  MoveL 8360 to (2.11, -17.65, -15.61) mm, rotated rx -180 ry 0 rz 0.01 deg; joints [33.024, -56.054, 126.414, -145.496, 74.243, 170.404]
  MoveL 8361 to (-4.42, -18.62, -15.85) mm, rotated rx 180 ry 0 rz 0.01 deg; joints [32.823, -55.856, 126.015, -145.669, 74.039, 170.344]
  MoveL 8362 to (-6.16, -24.99, -16.1) mm, rotated rx 180 ry 0 rz 0.01 deg; joints [32.532, -55.905, 126.173, -145.984, 74.074, 170.492]
  MoveL 8363 to (-1.01, -29.13, -16.34) mm, rotated rx 180 ry 0 rz 0.01 deg; joints [32.498, -56.122, 126.697, -146.066, 74.322, 170.68]
  MoveL 8364 to (4.84, -26.08, -16.58) mm, rotated rx 180 ry 0 rz 0.01 deg; joints [32.765, -56.228, 126.959, -145.819, 74.501, 170.695]
  MoveL 8365 to (4.39, -19.49, -16.83) mm, rotated rx -180 ry 0 rz 0.01 deg; joints [33.011, -56.076, 126.643, -145.542, 74.41, 170.529]
  MoveL 8366 to (-1.82, -17.26, -17.07) mm, rotated rx -180 ry 0 rz 0.01 deg; joints [32.941, -55.829, 126.127, -145.571, 74.176, 170.391]
  MoveL 8367 to (-6.36, -22.07, -17.32) mm, rotated rx -180 ry 0 rz 0.01 deg; joints [32.641, -55.764, 126.029, -145.871, 74.092, 170.459]
  MoveL 8368 to (-3.77, -28.14, -17.56) mm, rotated rx -180 ry 0 rz 0.01 deg; joints [32.469, -55.939, 126.464, -146.088, 74.276, 170.66]
  MoveL 8369 to (2.83, -28.21, -17.8) mm, rotated rx 180 ry 0 rz 0.01 deg; joints [32.632, -56.125, 126.912, -145.963, 74.522, 170.765]
  MoveL 8370 to (5.54, -22.19, -18.05) mm, rotated rx 180 ry 0 rz 0.01 deg; joints [32.936, -56.08, 126.832, -145.648, 74.55, 170.659]
  MoveL 8371 to (1.11, -17.29, -18.29) mm, rotated rx -180 ry 0 rz 0.01 deg; joints [33.014, -55.839, 126.321, -145.525, 74.342, 170.478]
  MoveL 8372 to (-5.16, -19.39, -18.54) mm, rotated rx -180 ry 0 rz 0.01 deg; joints [32.776, -55.671, 125.99, -145.743, 74.162, 170.451]
  MoveL 8373 to (-5.74, -25.97, -18.78) mm, rotated rx 180 ry 0 rz 0.01 deg; joints [32.506, -55.758, 126.234, -146.043, 74.241, 170.62]
  MoveL 8374 to (0.05, -29.14, -19.02) mm, rotated rx 180 ry 0 rz 0.01 deg; joints [32.526, -55.976, 126.76, -146.07, 74.5, 170.793]
  MoveL 8375 to (5.28, -25.1, -19.27) mm, rotated rx 180 ry 0 rz 0.01 deg; joints [32.816, -56.044, 126.937, -145.792, 74.643, 170.775]
  MoveL 8376 to (3.68, -18.7, -19.51) mm, rotated rx 180 ry 0 rz 0.01 deg; joints [33.025, -55.862, 126.55, -145.547, 74.514, 170.596]
  MoveL 8377 to (-2.84, -17.6, -19.76) mm, rotated rx 180 ry 0 rz 0.01 deg; joints [32.904, -55.628, 126.064, -145.63, 74.283, 170.483]
  MoveL 8378 to (-6.45, -23.13, -20) mm, rotated rx -180 ry 0 rz 0.01 deg; joints [32.6, -55.604, 126.058, -145.944, 74.241, 170.581]
  MoveC 8379 to (-4.81, -27.09, -20) mm, rotated rx 180 ry 0 rz 0.01 deg; joints [32.486, -55.726, 126.34, -146.085, 74.352, 170.706] to (-0.84, -28.73, -20) mm, rotated rx 180 ry 0 rz 0.01 deg; joints [32.521, -55.876, 126.678, -146.079, 74.514, 170.805]
  MoveC 8380 to (3.12, -27.09, -20) mm, rotated rx 180 ry 0 rz 0.01 deg; joints [32.684, -55.967, 126.875, -145.929, 74.632, 170.821] to (4.76, -23.13, -20) mm, rotated rx 180 ry 0 rz 0.01 deg; joints [32.881, -55.944, 126.814, -145.722, 74.637, 170.744]
  MoveL 8381 to (4.76, -20.36, -20) mm, rotated rx 180 ry 0 rz 0.01 deg; joints [32.989, -55.893, 126.694, -145.602, 74.6, 170.673]
  MoveC 8382 to (3.66, -18.8, -20) mm, rotated rx 180 ry 0 rz 0.01 deg; joints [33.021, -55.83, 126.551, -145.556, 74.54, 170.617] to (1.82, -19.33, -20) mm, rotated rx -180 ry 0 rz 0.01 deg; joints [32.954, -55.785, 126.451, -145.615, 74.482, 170.604]
  MoveL 8383 to (-0.78, -22.57, -20) mm, rotated rx -180 ry 0 rz 0.01 deg; joints [32.763, -55.766, 126.417, -145.808, 74.434, 170.649]
  MoveC 8384 to (-1.01, -24.64, -20) mm, rotated rx -180 ry 0 rz 0.01 deg; joints [32.676, -55.797, 126.491, -145.903, 74.454, 170.699] to (0.75, -25.75, -20) mm, rotated rx 180 ry 0 rz 0.01 deg; joints [32.677, -55.871, 126.658, -145.917, 74.531, 170.753]
  MoveL 8385 to (2.65, -25.75, -20) mm, rotated rx -180 ry 0 rz 0.01 deg; joints [32.725, -55.928, 126.785, -145.879, 74.598, 170.78]
  MoveC 8386 to (4.14, -25.13, -20) mm, rotated rx -180 ry 0 rz 0.01 deg; joints [32.787, -55.962, 126.859, -145.822, 74.642, 170.786] to (4.76, -23.64, -20) mm, rotated rx -180 ry 0 rz 0.01 deg; joints [32.861, -55.953, 126.836, -145.745, 74.644, 170.757]
  MoveL 8387 to (4.76, -23.13, -20) mm, rotated rx -180 ry 0 rz 0.01 deg; joints [32.881, -55.944, 126.814, -145.722, 74.637, 170.744]
  MoveL 8388 to (3.55, -23.39, -20) mm, rotated rx 180 ry 0 rz 0.01 deg; joints [32.84, -55.912, 126.744, -145.758, 74.598, 170.733]
  MoveL 8389 to (4.04, -24.46, -20) mm, rotated rx 180 ry 0 rz 0.01 deg; joints [32.81, -55.946, 126.823, -145.795, 74.629, 170.767]
  MoveL 8390 to (4.24, -24.7, -20) mm, rotated rx -180 ry 0 rz 0.01 deg; joints [32.806, -55.957, 126.847, -145.802, 74.64, 170.776]
  MoveL 8391 to (8.68, -28.03, -20) mm, rotated rx 180 ry 0 rz 0.01 deg; joints [32.788, -56.151, 127.288, -145.858, 74.841, 170.925]
  MoveL 8392 to (9.37, -28.67, -20) mm, rotated rx 180 ry 0 rz 0.01 deg; joints [32.78, -56.184, 127.362, -145.872, 74.873, 170.951]
  MoveL 8393 to (9.68, -28.6, -20) mm, rotated rx -180 ry 0 rz 0.01 deg; joints [32.79, -56.192, 127.38, -145.863, 74.883, 170.954]
  MoveL 8394 to (10.02, -27.8, -20) mm, rotated rx 180 ry 0 rz 0.01 deg; joints [32.831, -56.188, 127.368, -145.821, 74.885, 170.939]
  MoveL 8395 to (10.22, -26.94, -20) mm, rotated rx -180 ry 0 rz 0.01 deg; joints [32.869, -56.178, 127.344, -145.779, 74.88, 170.92]
  MoveL 8396 to (10.27, -25.87, -20) mm, rotated rx -180 ry 0 rz 0.01 deg; joints [32.913, -56.16, 127.302, -145.731, 74.868, 170.893]
  MoveL 8397 to (10.27, 7.5, -20) mm, rotated rx -180 ry 0 rz 0.01 deg; joints [34.203, -55.533, 125.827, -144.284, 74.418, 170.028]
  MoveL 8398 to (6.2, -2.89, -20) mm, rotated rx -180 ry 0 rz 0.01 deg; joints [33.701, -55.609, 126.021, -144.814, 74.416, 170.241]
  MoveL 8399 to (5.98, -3.35, -20) mm, rotated rx -180 ry 0 rz 0.01 deg; joints [33.678, -55.611, 126.027, -144.839, 74.414, 170.25]
  MoveL 8400 to (1.99, -10.24, -20) mm, rotated rx 180 ry 0 rz 0.01 deg; joints [33.311, -55.62, 126.065, -145.217, 74.367, 170.371]
  MoveL 8401 to (1.7, -10.66, -20) mm, rotated rx -180 ry 0 rz 0.01 deg; joints [33.287, -55.62, 126.064, -145.241, 74.362, 170.378]
  MoveL 8402 to (-6.19, -20.5, -20) mm, rotated rx 180 ry 0 rz 0.01 deg; joints [32.708, -55.563, 125.963, -145.824, 74.216, 170.518]
  MoveL 8403 to (-6.61, -20.95, -20) mm, rotated rx -180 ry 0 rz 0.01 deg; joints [32.68, -55.558, 125.953, -145.852, 74.206, 170.523]
  MoveL 8404 to (-7.35, -21.58, -20) mm, rotated rx -180 ry 0 rz 0.01 deg; joints [32.638, -55.548, 125.931, -145.894, 74.189, 170.529]
  MoveL 8405 to (-7.68, -21.83, -20) mm, rotated rx 180 ry 0 rz 0.01 deg; joints [32.619, -55.542, 125.919, -145.912, 74.18, 170.53]
  MoveL 8406 to (-17.93, -28.66, -20) mm, rotated rx 180 ry 0 rz 0.01 deg; joints [32.101, -55.353, 125.516, -146.407, 73.906, 170.558]
  MoveL 8407 to (-18.59, -29, -20) mm, rotated rx 180 ry 0 rz 0.01 deg; joints [32.072, -55.339, 125.486, -146.434, 73.887, 170.557]
  MoveL 8408 to (-19.94, -29.53, -20) mm, rotated rx 180 ry 0 rz 0.01 deg; joints [32.019, -55.307, 125.416, -146.482, 73.845, 170.551]
  MoveL 8409 to (-20.23, -29.62, -20) mm, rotated rx -180 ry 0 rz 0.01 deg; joints [32.008, -55.3, 125.401, -146.492, 73.836, 170.549]
  MoveL 8410 to (-25.91, -31.27, -20) mm, rotated rx 180 ry 0 rz 0.01 deg; joints [31.807, -55.153, 125.082, -146.67, 73.654, 170.51]
  MoveL 8411 to (5.41, -31.27, -20) mm, rotated rx 180 ry 0 rz 0.01 deg; joints [32.578, -56.112, 127.208, -146.066, 74.769, 170.96]
  MoveL 8412 to (6.62, -31.07, -20) mm, rotated rx 180 ry 0 rz 0.01 deg; joints [32.616, -56.145, 127.281, -146.033, 74.809, 170.972]
  MoveL 8413 to (7.44, -30.76, -20) mm, rotated rx -180 ry 0 rz 0.01 deg; joints [32.649, -56.164, 127.323, -146.003, 74.834, 170.976]
  MoveL 8414 to (7.66, -30.63, -20) mm, rotated rx 180 ry 0 rz 0.01 deg; joints [32.66, -56.168, 127.332, -145.992, 74.84, 170.976]
  MoveL 8415 to (7.91, -29.14, -20) mm, rotated rx 180 ry 0 rz 0.01 deg; joints [32.724, -56.148, 127.284, -145.922, 74.828, 170.942]
  MoveL 8416 to (5.43, -26.15, -20) mm, rotated rx 180 ry 0 rz 0.01 deg; joints [32.779, -56.019, 126.989, -145.841, 74.701, 170.83]
  MoveL 8417 to (5.26, -25.18, -20) mm, rotated rx 180 ry 0 rz 0.01 deg; joints [32.813, -55.996, 126.936, -145.802, 74.682, 170.803]
  MoveL 8418 to (3.73, -18.75, -20.24) mm, rotated rx 180 ry 0 rz 0.01 deg; joints [33.025, -55.816, 126.554, -145.554, 74.555, 170.626]
  MoveL 8419 to (-2.76, -17.57, -20.49) mm, rotated rx 180 ry 0 rz 0.01 deg; joints [32.908, -55.581, 126.065, -145.634, 74.323, 170.51]
  MoveL 8420 to (-6.45, -23.04, -20.73) mm, rotated rx -180 ry 0 rz 0.01 deg; joints [32.603, -55.554, 126.052, -145.947, 74.278, 170.606]
  MoveL 8421 to (-2.92, -28.62, -20.98) mm, rotated rx 180 ry 0 rz 0.01 deg; joints [32.474, -55.747, 126.53, -146.124, 74.49, 170.808]
  MoveL 8422 to (3.61, -27.62, -21.22) mm, rotated rx -180 ry 0 rz 0.01 deg; joints [32.676, -55.91, 126.925, -145.953, 74.72, 170.886]
  MoveL 8423 to (5.31, -21.25, -21.46) mm, rotated rx 180 ry 0 rz 0.01 deg; joints [32.969, -55.828, 126.763, -145.642, 74.707, 170.757]
  MoveL 8424 to (0.16, -17.12, -21.71) mm, rotated rx -180 ry 0 rz 0.01 deg; joints [32.999, -55.58, 126.237, -145.568, 74.483, 170.585]
  MoveL 8425 to (-5.69, -20.19, -21.95) mm, rotated rx 180 ry 0 rz 0.01 deg; joints [32.734, -55.444, 125.975, -145.819, 74.33, 170.587]
  MoveL 8426 to (-5.22, -26.78, -22.2) mm, rotated rx 180 ry 0 rz 0.01 deg; joints [32.489, -55.562, 126.29, -146.099, 74.447, 170.771]
  MoveL 8427 to (1, -28.99, -22.44) mm, rotated rx -180 ry 0 rz 0.01 deg; joints [32.558, -55.774, 126.804, -146.076, 74.71, 170.927]
  MoveL 8428 to (5.52, -24.19, -22.68) mm, rotated rx -180 ry 0 rz 0.01 deg; joints [32.86, -55.807, 126.9, -145.778, 74.818, 170.88]
  MoveL 8429 to (2.94, -18.12, -22.93) mm, rotated rx -180 ry 0 rz 0.01 deg; joints [33.032, -55.601, 126.462, -145.567, 74.657, 170.695]
  MoveL 8430 to (-3.66, -18.05, -23.17) mm, rotated rx -180 ry 0 rz 0.01 deg; joints [32.869, -55.385, 126.014, -145.697, 74.435, 170.606]
  MoveL 8431 to (-6.38, -24.06, -23.41) mm, rotated rx 180 ry 0 rz 0.01 deg; joints [32.567, -55.397, 126.09, -146.014, 74.433, 170.729]
  MoveL 8432 to (-1.95, -28.96, -23.66) mm, rotated rx -180 ry 0 rz 0.01 deg; joints [32.486, -55.603, 126.598, -146.144, 74.668, 170.927]
  MoveL 8433 to (4.31, -26.88, -23.9) mm, rotated rx -180 ry 0 rz 0.01 deg; joints [32.725, -55.737, 126.93, -145.93, 74.875, 170.974]
  MoveL 8434 to (4.91, -20.31, -24.15) mm, rotated rx 180 ry 0 rz 0.01 deg; joints [32.997, -55.62, 126.685, -145.634, 74.819, 170.825]
  MoveL 8435 to (-0.86, -17.11, -24.39) mm, rotated rx 180 ry 0 rz 0.01 deg; joints [32.976, -55.372, 126.157, -145.612, 74.584, 170.667]
  MoveL 8436 to (-6.11, -21.12, -24.63) mm, rotated rx 180 ry 0 rz 0.01 deg; joints [32.689, -55.271, 125.976, -145.892, 74.465, 170.702]
  MoveL 8437 to (-4.54, -27.54, -24.88) mm, rotated rx 180 ry 0 rz 0.01 deg; joints [32.479, -55.418, 126.358, -146.143, 74.621, 170.897]
  MoveL 8438 to (1.96, -28.67, -25.12) mm, rotated rx 180 ry 0 rz 0.01 deg; joints [32.597, -55.618, 126.844, -146.066, 74.88, 171.03]
  MoveL 8439 to (5.62, -23.17, -25.37) mm, rotated rx -180 ry 0 rz 0.01 deg; joints [32.904, -55.611, 126.851, -145.755, 74.947, 170.953]
  MoveL 8440 to (2.04, -17.62, -25.61) mm, rotated rx 180 ry 0 rz 0.01 deg; joints [33.03, -55.387, 126.369, -145.587, 74.757, 170.767]
  MoveL 8441 to (-4.47, -18.67, -25.85) mm, rotated rx 180 ry 0 rz 0.01 deg; joints [32.826, -55.195, 125.975, -145.764, 74.552, 170.706]
  MoveL 8442 to (-6.13, -25.05, -26.1) mm, rotated rx -180 ry 0 rz 0.01 deg; joints [32.537, -55.245, 126.138, -146.077, 74.593, 170.854]
  MoveL 8443 to (-0.95, -29.14, -26.34) mm, rotated rx 180 ry 0 rz 0.01 deg; joints [32.506, -55.457, 126.662, -146.155, 74.846, 171.042]
  MoveL 8444 to (4.87, -26.03, -26.59) mm, rotated rx 180 ry 0 rz 0.01 deg; joints [32.774, -55.559, 126.919, -145.905, 75.023, 171.058]
  MoveL 8445 to (4.36, -19.45, -26.83) mm, rotated rx 180 ry 0 rz 0.01 deg; joints [33.019, -55.408, 126.599, -145.631, 74.927, 170.892]
  MoveL 8446 to (-1.87, -17.28, -27.07) mm, rotated rx -180 ry 0 rz 0.01 deg; joints [32.946, -55.166, 126.084, -145.663, 74.688, 170.753]
  MoveL 8447 to (-6.36, -22.11, -27.32) mm, rotated rx -180 ry 0 rz 0.01 deg; joints [32.646, -55.104, 125.99, -145.964, 74.607, 170.819]
  MoveL 8448 to (-3.74, -28.17, -27.56) mm, rotated rx 180 ry 0 rz 0.01 deg; joints [32.476, -55.275, 126.427, -146.178, 74.797, 171.02]
  MoveL 8449 to (2.87, -28.19, -27.8) mm, rotated rx 180 ry 0 rz 0.01 deg; joints [32.64, -55.456, 126.872, -146.051, 75.045, 171.127]
  MoveL 8450 to (5.54, -22.15, -28.05) mm, rotated rx -180 ry 0 rz 0.01 deg; joints [32.944, -55.411, 126.789, -145.736, 75.069, 171.023]
  MoveL 8451 to (1.08, -17.29, -28.29) mm, rotated rx -180 ry 0 rz 0.01 deg; joints [33.021, -55.174, 126.277, -145.616, 74.856, 170.841]
  MoveL 8452 to (-5.17, -19.41, -28.54) mm, rotated rx -180 ry 0 rz 0.01 deg; joints [32.781, -55.01, 125.948, -145.834, 74.675, 170.811]
  MoveL 8453 to (-5.73, -25.99, -28.78) mm, rotated rx -180 ry 0 rz 0.01 deg; joints [32.512, -55.095, 126.193, -146.133, 74.759, 170.979]
  MoveL 8454 to (0.07, -29.14, -29.02) mm, rotated rx -180 ry 0 rz 0.01 deg; joints [32.534, -55.308, 126.719, -146.158, 75.022, 171.154]
  MoveL 8455 to (5.29, -25.09, -29.27) mm, rotated rx -180 ry 0 rz 0.01 deg; joints [32.823, -55.374, 126.894, -145.88, 75.164, 171.138]
  MoveL 8456 to (3.67, -18.69, -29.51) mm, rotated rx 180 ry 0 rz 0.01 deg; joints [33.032, -55.195, 126.507, -145.636, 75.03, 170.96]
  MoveL 8457 to (-2.84, -17.6, -29.76) mm, rotated rx -180 ry 0 rz 0.01 deg; joints [32.911, -54.966, 126.021, -145.72, 74.796, 170.843]
  MoveL 8458 to (-6.45, -23.13, -30) mm, rotated rx -180 ry 0 rz 0.01 deg; joints [32.606, -54.941, 126.016, -146.033, 74.756, 170.939]
  MoveC 8459 to (-0.84, -28.74, -30) mm, rotated rx 180 ry 0 rz 0.01 deg; joints [32.527, -55.209, 126.635, -146.167, 75.034, 171.165] to (4.76, -23.13, -30) mm, rotated rx -180 ry 0 rz 0.01 deg; joints [32.887, -55.275, 126.771, -145.811, 75.156, 171.107]
  MoveL 8460 to (4.76, -20.36, -30) mm, rotated rx -180 ry 0 rz 0.01 deg; joints [32.995, -55.225, 126.651, -145.69, 75.117, 171.036]
  MoveC 8461 to (3.66, -18.8, -30) mm, rotated rx -180 ry 0 rz 0.01 deg; joints [33.028, -55.164, 126.509, -145.645, 75.056, 170.98] to (1.82, -19.33, -30) mm, rotated rx -180 ry 0 rz 0.01 deg; joints [32.961, -55.119, 126.408, -145.705, 74.998, 170.966]
  MoveL 8462 to (-0.77, -22.57, -30) mm, rotated rx 180 ry 0 rz 0.01 deg; joints [32.77, -55.1, 126.374, -145.897, 74.951, 171.01]
  MoveC 8463 to (-1.01, -24.64, -30) mm, rotated rx 180 ry 0 rz 0.01 deg; joints [32.683, -55.131, 126.448, -145.992, 74.971, 171.059] to (0.76, -25.75, -30) mm, rotated rx 180 ry 0 rz 0.01 deg; joints [32.684, -55.203, 126.615, -146.005, 75.05, 171.113]
  MoveL 8464 to (2.65, -25.75, -30) mm, rotated rx -180 ry 0 rz 0.01 deg; joints [32.731, -55.259, 126.742, -145.967, 75.117, 171.141]
  MoveC 8465 to (4.14, -25.14, -30) mm, rotated rx -180 ry 0 rz 0.01 deg; joints [32.793, -55.292, 126.816, -145.911, 75.162, 171.148] to (4.76, -23.64, -30) mm, rotated rx -180 ry 0 rz 0.01 deg; joints [32.867, -55.284, 126.793, -145.833, 75.163, 171.119]
  MoveL 8466 to (4.76, -23.13, -30) mm, rotated rx 180 ry 0 rz 0.01 deg; joints [32.887, -55.275, 126.771, -145.811, 75.156, 171.107]
  MoveL 8467 to (3.55, -23.4, -30) mm, rotated rx 180 ry 0 rz 0.01 deg; joints [32.846, -55.244, 126.701, -145.847, 75.116, 171.095]
  MoveL 8468 to (4.04, -24.46, -30) mm, rotated rx 180 ry 0 rz 0.01 deg; joints [32.817, -55.277, 126.78, -145.883, 75.149, 171.13]
  MoveL 8469 to (4.24, -24.7, -30) mm, rotated rx -180 ry 0 rz 0.01 deg; joints [32.813, -55.287, 126.804, -145.89, 75.159, 171.139]
  MoveL 8470 to (8.68, -28.03, -30) mm, rotated rx -180 ry 0 rz 0.01 deg; joints [32.794, -55.478, 127.245, -145.945, 75.364, 171.289]
  MoveL 8471 to (9.37, -28.67, -30) mm, rotated rx 180 ry 0 rz 0.01 deg; joints [32.787, -55.509, 127.318, -145.959, 75.397, 171.315]
  MoveL 8472 to (9.68, -28.6, -30) mm, rotated rx 180 ry 0 rz 0.01 deg; joints [32.797, -55.517, 127.336, -145.95, 75.407, 171.318]
  MoveL 8473 to (10.02, -27.8, -30) mm, rotated rx 180 ry 0 rz 0.01 deg; joints [32.837, -55.513, 127.325, -145.908, 75.408, 171.303]
  MoveL 8474 to (10.22, -26.94, -30) mm, rotated rx 180 ry 0 rz 0.01 deg; joints [32.876, -55.504, 127.301, -145.866, 75.403, 171.284]
  MoveL 8475 to (10.27, -25.87, -30) mm, rotated rx -180 ry 0 rz 0.01 deg; joints [32.92, -55.486, 127.258, -145.819, 75.39, 171.258]
  MoveL 8476 to (10.27, 7.47, -30) mm, rotated rx -180 ry 0 rz 0.01 deg; joints [34.208, -54.873, 125.786, -144.378, 74.921, 170.4]
  MoveL 8477 to (6.2, -2.89, -30) mm, rotated rx -180 ry 0 rz 0.01 deg; joints [33.707, -54.947, 125.978, -144.906, 74.923, 170.609]
  MoveL 8478 to (5.98, -3.35, -30) mm, rotated rx -180 ry 0 rz 0.01 deg; joints [33.684, -54.949, 125.984, -144.93, 74.922, 170.617]
  MoveL 8479 to (1.99, -10.24, -30) mm, rotated rx -180 ry 0 rz 0.01 deg; joints [33.317, -54.958, 126.022, -145.308, 74.877, 170.735]
  MoveL 8480 to (1.7, -10.66, -30) mm, rotated rx 180 ry 0 rz 0.01 deg; joints [33.294, -54.957, 126.021, -145.331, 74.873, 170.742]
  MoveL 8481 to (-6.17, -20.5, -30) mm, rotated rx -180 ry 0 rz 0.01 deg; joints [32.715, -54.902, 125.92, -145.914, 74.729, 170.876]
  MoveL 8482 to (-6.62, -20.95, -30) mm, rotated rx 180 ry 0 rz 0.01 deg; joints [32.687, -54.897, 125.91, -145.942, 74.72, 170.881]
  MoveL 8483 to (-7.36, -21.59, -30) mm, rotated rx 180 ry 0 rz 0.01 deg; joints [32.644, -54.887, 125.888, -145.984, 74.702, 170.886]
  MoveL 8484 to (-7.67, -21.83, -30) mm, rotated rx 180 ry 0 rz 0.01 deg; joints [32.626, -54.881, 125.877, -146.001, 74.694, 170.888]
  MoveL 8485 to (-17.71, -28.55, -30) mm, rotated rx 180 ry 0 rz 0.01 deg; joints [32.118, -54.7, 125.484, -146.487, 74.426, 170.909]
  MoveL 8486 to (-18.19, -28.82, -30) mm, rotated rx 180 ry 0 rz 0.01 deg; joints [32.096, -54.691, 125.463, -146.508, 74.412, 170.909]
  MoveL 8487 to (-19.2, -29.28, -30) mm, rotated rx 180 ry 0 rz 0.01 deg; joints [32.054, -54.668, 125.414, -146.547, 74.382, 170.906]
  MoveL 8488 to (-19.64, -29.44, -30) mm, rotated rx 180 ry 0 rz 0.01 deg; joints [32.036, -54.658, 125.391, -146.563, 74.368, 170.903]
  MoveL 8489 to (-25.81, -31.27, -30) mm, rotated rx -180 ry 0 rz 0.01 deg; joints [31.816, -54.503, 125.046, -146.758, 74.17, 170.858]
  MoveL 8490 to (5.41, -31.27, -30) mm, rotated rx 180 ry 0 rz 0.01 deg; joints [32.585, -55.439, 127.165, -146.153, 75.293, 171.321]
  MoveL 8491 to (6.62, -31.07, -30) mm, rotated rx 180 ry 0 rz 0.01 deg; joints [32.623, -55.471, 127.238, -146.12, 75.333, 171.335]
  MoveL 8492 to (7.44, -30.76, -30) mm, rotated rx 180 ry 0 rz 0.01 deg; joints [32.656, -55.49, 127.28, -146.09, 75.358, 171.339]
  MoveL 8493 to (7.66, -30.63, -30) mm, rotated rx -180 ry 0 rz 0.01 deg; joints [32.667, -55.494, 127.288, -146.079, 75.364, 171.339]
  MoveL 8494 to (7.91, -29.14, -30) mm, rotated rx -180 ry 0 rz 0.01 deg; joints [32.731, -55.475, 127.241, -146.009, 75.352, 171.305]
  MoveL 8495 to (5.43, -26.15, -30) mm, rotated rx -180 ry 0 rz 0.01 deg; joints [32.786, -55.348, 126.946, -145.929, 75.222, 171.193]
  MoveL 8496 to (5.26, -25.18, -30) mm, rotated rx 180 ry 0 rz 0.01 deg; joints [32.82, -55.326, 126.893, -145.89, 75.202, 171.166]
  MoveL 8497 to (3.74, -18.75, -30.24) mm, rotated rx 180 ry 0 rz 0.01 deg; joints [33.032, -55.149, 126.511, -145.643, 75.071, 170.989]
  MoveL 8498 to (-2.76, -17.57, -30.49) mm, rotated rx 180 ry 0 rz 0.01 deg; joints [32.914, -54.919, 126.022, -145.724, 74.835, 170.87]
  MoveL 8499 to (-6.45, -23.05, -30.73) mm, rotated rx -180 ry 0 rz 0.01 deg; joints [32.61, -54.891, 126.009, -146.036, 74.792, 170.963]
  MoveL 8500 to (-2.92, -28.62, -30.98) mm, rotated rx -180 ry 0 rz 0.01 deg; joints [32.481, -55.08, 126.486, -146.211, 75.009, 171.165]
  MoveL 8501 to (3.61, -27.62, -31.22) mm, rotated rx -180 ry 0 rz 0.01 deg; joints [32.683, -55.239, 126.881, -146.04, 75.241, 171.247]
  MoveL 8502 to (5.31, -21.25, -31.46) mm, rotated rx 180 ry 0 rz 0.01 deg; joints [32.976, -55.159, 126.719, -145.73, 75.224, 171.12]
  MoveL 8503 to (0.16, -17.13, -31.71) mm, rotated rx 180 ry 0 rz 0.01 deg; joints [33.006, -54.916, 126.192, -145.657, 74.996, 170.946]
  MoveL 8504 to (-5.69, -20.19, -31.95) mm, rotated rx -180 ry 0 rz 0.01 deg; joints [32.741, -54.782, 125.931, -145.908, 74.842, 170.945]
  MoveL 8505 to (-5.22, -26.78, -32.2) mm, rotated rx 180 ry 0 rz 0.01 deg; joints [32.496, -54.897, 126.245, -146.187, 74.963, 171.128]
  MoveL 8506 to (1, -29, -32.44) mm, rotated rx 180 ry 0 rz 0.01 deg; joints [32.565, -55.104, 126.759, -146.163, 75.23, 171.286]
  MoveL 8507 to (5.52, -24.19, -32.68) mm, rotated rx 180 ry 0 rz 0.01 deg; joints [32.867, -55.136, 126.854, -145.865, 75.336, 171.241]
  MoveL 8508 to (2.94, -18.12, -32.93) mm, rotated rx -180 ry 0 rz 0.01 deg; joints [33.038, -54.935, 126.416, -145.655, 75.171, 171.057]
  MoveL 8509 to (-3.66, -18.05, -33.17) mm, rotated rx 180 ry 0 rz 0.01 deg; joints [32.875, -54.722, 125.968, -145.785, 74.947, 170.964]
  MoveL 8510 to (-6.38, -24.06, -33.41) mm, rotated rx 180 ry 0 rz 0.01 deg; joints [32.574, -54.733, 126.044, -146.102, 74.946, 171.085]
  MoveL 8511 to (-1.95, -28.96, -33.66) mm, rotated rx 180 ry 0 rz 0.01 deg; joints [32.493, -54.935, 126.552, -146.23, 75.187, 171.284]
  MoveL 8512 to (4.31, -26.88, -33.9) mm, rotated rx -180 ry 0 rz 0.01 deg; joints [32.732, -55.066, 126.883, -146.016, 75.394, 171.335]
  MoveL 8513 to (4.91, -20.31, -34.15) mm, rotated rx 180 ry 0 rz 0.01 deg; joints [33.004, -54.95, 126.638, -145.72, 75.335, 171.187]
  MoveL 8514 to (-0.86, -17.12, -34.39) mm, rotated rx -180 ry 0 rz 0.01 deg; joints [32.982, -54.707, 126.11, -145.7, 75.096, 171.026]
  MoveL 8515 to (-6.11, -21.13, -34.63) mm, rotated rx -180 ry 0 rz 0.01 deg; joints [32.696, -54.608, 125.929, -145.98, 74.977, 171.058]
  MoveL 8516 to (-4.54, -27.54, -34.88) mm, rotated rx -180 ry 0 rz 0.01 deg; joints [32.485, -54.752, 126.31, -146.229, 75.137, 171.252]
  MoveL 8517 to (1.97, -28.67, -35.12) mm, rotated rx 180 ry 0 rz 0.01 deg; joints [32.603, -54.947, 126.796, -146.152, 75.399, 171.388]
  MoveL 8518 to (5.62, -23.17, -35.37) mm, rotated rx 180 ry 0 rz 0.01 deg; joints [32.911, -54.94, 126.803, -145.841, 75.464, 171.313]
  MoveL 8519 to (2.04, -17.62, -35.61) mm, rotated rx 180 ry 0 rz 0.01 deg; joints [33.037, -54.72, 126.321, -145.674, 75.269, 171.127]
  MoveL 8520 to (-4.47, -18.67, -35.85) mm, rotated rx -180 ry 0 rz 0.01 deg; joints [32.833, -54.531, 125.927, -145.851, 75.063, 171.063]
  MoveL 8521 to (-6.13, -25.06, -36.1) mm, rotated rx 180 ry 0 rz 0.01 deg; joints [32.543, -54.579, 126.089, -146.163, 75.106, 171.208]
  MoveL 8522 to (-0.95, -29.14, -36.34) mm, rotated rx 180 ry 0 rz 0.01 deg; joints [32.513, -54.787, 126.614, -146.24, 75.364, 171.398]
  MoveL 8523 to (4.87, -26.03, -36.59) mm, rotated rx 180 ry 0 rz 0.01 deg; joints [32.781, -54.886, 126.87, -145.99, 75.541, 171.418]
  MoveL 8524 to (4.36, -19.45, -36.83) mm, rotated rx 180 ry 0 rz 0.01 deg; joints [33.025, -54.739, 126.549, -145.717, 75.44, 171.253]
  MoveL 8525 to (-1.87, -17.28, -37.07) mm, rotated rx 180 ry 0 rz 0.01 deg; joints [32.953, -54.501, 126.035, -145.75, 75.198, 171.111]
  MoveL 8526 to (-6.36, -22.11, -37.32) mm, rotated rx 180 ry 0 rz 0.01 deg; joints [32.653, -54.439, 125.941, -146.05, 75.118, 171.173]
  MoveL 8527 to (-3.73, -28.17, -37.56) mm, rotated rx 180 ry 0 rz 0.01 deg; joints [32.482, -54.607, 126.377, -146.263, 75.312, 171.375]
  MoveL 8528 to (2.87, -28.19, -37.8) mm, rotated rx -180 ry 0 rz 0.01 deg; joints [32.647, -54.784, 126.822, -146.135, 75.563, 171.484]
  MoveL 8529 to (5.54, -22.16, -38.05) mm, rotated rx -180 ry 0 rz 0.01 deg; joints [32.95, -54.739, 126.739, -145.821, 75.584, 171.383]
  MoveL 8530 to (1.08, -17.29, -38.29) mm, rotated rx -180 ry 0 rz 0.01 deg; joints [33.027, -54.506, 126.227, -145.702, 75.366, 171.2]
  MoveL 8531 to (-5.17, -19.42, -38.54) mm, rotated rx -180 ry 0 rz 0.01 deg; joints [32.788, -54.345, 125.898, -145.92, 75.185, 171.166]
  MoveL 8532 to (-5.73, -25.99, -38.78) mm, rotated rx -180 ry 0 rz 0.01 deg; joints [32.519, -54.429, 126.143, -146.218, 75.272, 171.332]
  MoveL 8533 to (0.07, -29.14, -39.02) mm, rotated rx -180 ry 0 rz 0.01 deg; joints [32.54, -54.637, 126.668, -146.242, 75.539, 171.509]
  MoveL 8534 to (5.29, -25.1, -39.27) mm, rotated rx 180 ry 0 rz 0.01 deg; joints [32.83, -54.701, 126.843, -145.963, 75.68, 171.496]
  MoveL 8535 to (3.67, -18.7, -39.51) mm, rotated rx -180 ry 0 rz 0.01 deg; joints [33.039, -54.525, 126.456, -145.721, 75.542, 171.319]
  MoveL 8536 to (-2.84, -17.61, -39.76) mm, rotated rx 180 ry 0 rz 0.01 deg; joints [32.917, -54.3, 125.97, -145.806, 75.305, 171.199]
  MoveL 8537 to (-6.45, -23.13, -40) mm, rotated rx 180 ry 0 rz 0.01 deg; joints [32.613, -54.276, 125.964, -146.118, 75.266, 171.292]
  MoveC 8538 to (-0.84, -28.74, -40) mm, rotated rx 180 ry 0 rz 0.01 deg; joints [32.534, -54.537, 126.583, -146.251, 75.55, 171.519] to (4.76, -23.13, -40) mm, rotated rx 180 ry 0 rz 0.01 deg; joints [32.894, -54.602, 126.719, -145.895, 75.671, 171.465]
  MoveL 8539 to (4.76, -20.36, -40) mm, rotated rx -180 ry 0 rz 0.01 deg; joints [33.002, -54.553, 126.599, -145.775, 75.63, 171.395]
  MoveC 8540 to (3.66, -18.8, -40) mm, rotated rx -180 ry 0 rz 0.01 deg; joints [33.035, -54.494, 126.457, -145.729, 75.568, 171.339] to (1.82, -19.33, -40) mm, rotated rx 180 ry 0 rz 0.01 deg; joints [32.968, -54.45, 126.356, -145.789, 75.509, 171.323]
  MoveL 8541 to (-0.77, -22.57, -40) mm, rotated rx -180 ry 0 rz 0.01 deg; joints [32.777, -54.432, 126.323, -145.981, 75.463, 171.365]
  MoveC 8542 to (-1.01, -24.64, -40) mm, rotated rx -180 ry 0 rz 0.01 deg; joints [32.69, -54.461, 126.396, -146.076, 75.485, 171.414] to (0.76, -25.76, -40) mm, rotated rx -180 ry 0 rz 0.01 deg; joints [32.691, -54.532, 126.563, -146.089, 75.565, 171.469]
  MoveL 8543 to (2.65, -25.76, -40) mm, rotated rx 180 ry 0 rz 0.01 deg; joints [32.738, -54.587, 126.69, -146.051, 75.633, 171.498]
  MoveC 8544 to (4.15, -25.14, -40) mm, rotated rx 180 ry 0 rz 0.01 deg; joints [32.8, -54.619, 126.764, -145.994, 75.678, 171.505] to (4.76, -23.64, -40) mm, rotated rx 180 ry 0 rz 0.01 deg; joints [32.874, -54.611, 126.741, -145.917, 75.678, 171.478]
  MoveL 8545 to (4.76, -23.13, -40) mm, rotated rx -180 ry 0 rz 0.01 deg; joints [32.894, -54.602, 126.719, -145.895, 75.671, 171.465]
  MoveL 8546 to (3.55, -23.4, -40) mm, rotated rx 180 ry 0 rz 0.01 deg; joints [32.853, -54.572, 126.649, -145.931, 75.631, 171.453]
  MoveL 8547 to (4.04, -24.46, -40) mm, rotated rx 180 ry 0 rz 0.01 deg; joints [32.824, -54.605, 126.728, -145.967, 75.664, 171.487]
  MoveL 8548 to (4.24, -24.7, -40) mm, rotated rx -180 ry 0 rz 0.01 deg; joints [32.819, -54.614, 126.752, -145.973, 75.675, 171.496]
  MoveL 8549 to (8.68, -28.03, -40) mm, rotated rx -180 ry 0 rz 0.01 deg; joints [32.801, -54.801, 127.192, -146.028, 75.883, 171.648]
  MoveL 8550 to (9.37, -28.67, -40) mm, rotated rx -180 ry 0 rz 0.01 deg; joints [32.793, -54.832, 127.266, -146.042, 75.917, 171.674]
  MoveL 8551 to (9.68, -28.6, -40) mm, rotated rx 180 ry 0 rz 0.01 deg; joints [32.804, -54.839, 127.284, -146.033, 75.927, 171.677]
  MoveL 8552 to (10.02, -27.8, -40) mm, rotated rx 180 ry 0 rz 0.01 deg; joints [32.844, -54.835, 127.273, -145.991, 75.928, 171.663]
  MoveL 8553 to (10.22, -26.94, -40) mm, rotated rx 180 ry 0 rz 0.01 deg; joints [32.883, -54.826, 127.249, -145.949, 75.922, 171.644]
  MoveL 8554 to (10.27, -25.87, -40) mm, rotated rx 180 ry 0 rz 0.01 deg; joints [32.926, -54.809, 127.206, -145.901, 75.908, 171.618]
  MoveL 8555 to (10.27, 7.44, -40) mm, rotated rx 180 ry 0 rz 0.01 deg; joints [34.214, -54.21, 125.736, -144.467, 75.42, 170.767]
  MoveL 8556 to (6.19, -2.89, -40) mm, rotated rx 180 ry 0 rz 0.01 deg; joints [33.714, -54.282, 125.927, -144.993, 75.427, 170.972]
  MoveL 8557 to (5.98, -3.35, -40) mm, rotated rx 180 ry 0 rz 0.01 deg; joints [33.691, -54.284, 125.932, -145.016, 75.425, 170.98]
  MoveL 8558 to (1.99, -10.24, -40) mm, rotated rx -180 ry 0 rz 0.01 deg; joints [33.324, -54.293, 125.97, -145.394, 75.383, 171.095]
  MoveL 8559 to (1.7, -10.66, -40) mm, rotated rx 180 ry 0 rz 0.01 deg; joints [33.3, -54.292, 125.969, -145.417, 75.379, 171.101]
  MoveL 8560 to (-6.17, -20.49, -40) mm, rotated rx 180 ry 0 rz 0.01 deg; joints [32.722, -54.238, 125.869, -145.999, 75.239, 171.23]
  MoveL 8561 to (-6.61, -20.95, -40) mm, rotated rx 180 ry 0 rz 0.01 deg; joints [32.693, -54.233, 125.859, -146.027, 75.229, 171.234]
  MoveL 8562 to (-7.36, -21.59, -40) mm, rotated rx -180 ry 0 rz 0.01 deg; joints [32.65, -54.222, 125.836, -146.07, 75.211, 171.239]
  MoveL 8563 to (-7.67, -21.82, -40) mm, rotated rx -180 ry 0 rz 0.01 deg; joints [32.633, -54.217, 125.825, -146.086, 75.204, 171.24]
  MoveL 8564 to (-17.48, -28.43, -40) mm, rotated rx 180 ry 0 rz 0.01 deg; joints [32.135, -54.044, 125.443, -146.563, 74.942, 171.257]
  MoveL 8565 to (-17.94, -28.7, -40) mm, rotated rx -180 ry 0 rz 0.01 deg; joints [32.113, -54.035, 125.423, -146.583, 74.929, 171.256]
  MoveL 8566 to (-19.17, -29.27, -40) mm, rotated rx 180 ry 0 rz 0.01 deg; joints [32.061, -54.009, 125.363, -146.631, 74.892, 171.252]
  MoveL 8567 to (-19.62, -29.44, -40) mm, rotated rx -180 ry 0 rz 0.01 deg; joints [32.044, -53.998, 125.34, -146.647, 74.878, 171.249]
  MoveL 8568 to (-25.71, -31.27, -40) mm, rotated rx 180 ry 0 rz 0.01 deg; joints [31.825, -53.849, 125.002, -146.842, 74.681, 171.202]
  MoveL 8569 to (5.41, -31.27, -40) mm, rotated rx -180 ry 0 rz 0.01 deg; joints [32.591, -54.763, 127.112, -146.235, 75.812, 171.678]
  MoveL 8570 to (6.62, -31.07, -40) mm, rotated rx 180 ry 0 rz 0.01 deg; joints [32.629, -54.794, 127.185, -146.202, 75.853, 171.692]
  MoveL 8571 to (7.44, -30.76, -40) mm, rotated rx 180 ry 0 rz 0.01 deg; joints [32.662, -54.813, 127.227, -146.172, 75.878, 171.697]
  MoveL 8572 to (7.66, -30.63, -40) mm, rotated rx -180 ry 0 rz 0.01 deg; joints [32.673, -54.817, 127.236, -146.162, 75.884, 171.697]
  MoveL 8573 to (7.67, -29.55, -40) mm, rotated rx -180 ry 0 rz 0.01 deg; joints [32.716, -54.798, 127.191, -146.115, 75.869, 171.67]
  MoveL 8574 to (3.92, -27.15, -40) mm, rotated rx -180 ry 0 rz 0.01 deg; joints [32.715, -54.648, 126.835, -146.086, 75.699, 171.552]
  MoveL 8575 to (-0.53, -24.82, -40) mm, rotated rx 180 ry 0 rz 0.01 deg; joints [32.695, -54.478, 126.436, -146.074, 75.505, 171.426]
  MoveL 8576 to (-1.53, -24.26, -40) mm, rotated rx -180 ry 0 rz 0.01 deg; joints [32.692, -54.439, 126.344, -146.07, 75.46, 171.396]
  MoveL 8577 to (-1.89, -24.46, -40) mm, rotated rx 180 ry 0 rz 0.01 deg; joints [32.675, -54.432, 126.329, -146.086, 75.45, 171.395]
  MoveL 8578 to (1.29, -30.05, -40.24) mm, rotated rx 180 ry 0 rz 0.01 deg; joints [32.536, -54.606, 126.782, -146.267, 75.658, 171.593]
  MoveL 8579 to (7.7, -29.59, -40.47) mm, rotated rx 180 ry 0 rz 0.01 deg; joints [32.715, -54.768, 127.192, -146.12, 75.895, 171.689]
  MoveL 8580 to (10.06, -23.61, -40.71) mm, rotated rx 180 ry 0 rz 0.01 deg; joints [33.01, -54.715, 127.09, -145.813, 75.904, 171.584]
  MoveL 8581 to (5.69, -18.9, -40.95) mm, rotated rx 180 ry 0 rz 0.01 deg; joints [33.083, -54.49, 126.591, -145.7, 75.69, 171.406]
  MoveL 8582 to (-0.45, -20.81, -41.18) mm, rotated rx 180 ry 0 rz 0.01 deg; joints [32.854, -54.33, 126.261, -145.909, 75.51, 171.368]
  MoveL 8583 to (-1.38, -27.17, -41.42) mm, rotated rx 180 ry 0 rz 0.01 deg; joints [32.583, -54.399, 126.472, -146.205, 75.581, 171.521]
  MoveL 8584 to (3.96, -30.76, -41.66) mm, rotated rx 180 ry 0 rz 0.01 deg; joints [32.576, -54.6, 126.984, -146.256, 75.838, 171.702]
  MoveL 8585 to (9.5, -27.49, -41.89) mm, rotated rx -180 ry 0 rz 0.01 deg; joints [32.844, -54.686, 127.213, -146.003, 76.002, 171.715]
  MoveL 8586 to (8.94, -21.08, -42.13) mm, rotated rx 180 ry 0 rz 0.01 deg; joints [33.081, -54.542, 126.897, -145.738, 75.9, 171.554]
  MoveL 8587 to (2.92, -18.82, -42.37) mm, rotated rx 180 ry 0 rz 0.01 deg; joints [33.017, -54.314, 126.394, -145.764, 75.662, 171.412]
  MoveL 8588 to (-1.72, -23.27, -42.61) mm, rotated rx -180 ry 0 rz 0.01 deg; joints [32.727, -54.242, 126.274, -146.052, 75.572, 171.46]
  MoveL 8589 to (0.29, -29.38, -42.84) mm, rotated rx 180 ry 0 rz 0.01 deg; joints [32.539, -54.39, 126.671, -146.279, 75.746, 171.652]
  MoveL 8590 to (6.67, -30.2, -43.08) mm, rotated rx -180 ry 0 rz 0.01 deg; joints [32.667, -54.571, 127.133, -146.188, 76.001, 171.78]
  MoveL 8591 to (10.17, -24.81, -43.32) mm, rotated rx 180 ry 0 rz 0.01 deg; joints [32.967, -54.562, 127.134, -145.884, 76.06, 171.709]
  MoveL 8592 to (6.81, -19.32, -43.55) mm, rotated rx -180 ry 0 rz 0.01 deg; joints [33.097, -54.354, 126.67, -145.717, 75.87, 171.527]
  MoveL 8593 to (0.41, -19.98, -43.79) mm, rotated rx 180 ry 0 rz 0.01 deg; joints [32.91, -54.166, 126.268, -145.877, 75.661, 171.452]
  MoveL 8594 to (-1.75, -26.03, -44.03) mm, rotated rx -180 ry 0 rz 0.01 deg; joints [32.62, -54.193, 126.382, -146.184, 75.684, 171.579]
  MoveL 8595 to (2.77, -30.6, -44.26) mm, rotated rx 180 ry 0 rz 0.01 deg; joints [32.554, -54.386, 126.882, -146.294, 75.927, 171.771]
  MoveL 8596 to (8.85, -28.5, -44.5) mm, rotated rx -180 ry 0 rz 0.01 deg; joints [32.79, -54.508, 127.197, -146.081, 76.128, 171.822]
  MoveC 8597 to (7.97, -20.62, -44.5) mm, rotated rx 180 ry 0 rz 0.01 deg; joints [33.076, -54.346, 126.798, -145.757, 75.979, 171.612] to (0.09, -21.49, -44.5) mm, rotated rx -180 ry 0 rz 0.01 deg; joints [32.843, -54.135, 126.308, -145.954, 75.708, 171.51]
  MoveL 8598 to (-0.77, -22.57, -44.5) mm, rotated rx 180 ry 0 rz 0.01 deg; joints [32.78, -54.129, 126.296, -146.018, 75.692, 171.524]
  MoveC 8599 to (-1.01, -24.64, -44.5) mm, rotated rx 180 ry 0 rz 0.01 deg; joints [32.693, -54.159, 126.37, -146.113, 75.714, 171.572] to (0.76, -25.75, -44.5) mm, rotated rx 180 ry 0 rz 0.01 deg; joints [32.694, -54.229, 126.537, -146.125, 75.795, 171.627]
  MoveL 8600 to (2.65, -25.75, -44.5) mm, rotated rx 180 ry 0 rz 0.01 deg; joints [32.741, -54.283, 126.664, -146.087, 75.863, 171.657]
  MoveC 8601 to (4.14, -25.14, -44.5) mm, rotated rx 180 ry 0 rz 0.01 deg; joints [32.803, -54.315, 126.737, -146.03, 75.908, 171.665] to (4.76, -23.64, -44.5) mm, rotated rx 180 ry 0 rz 0.01 deg; joints [32.877, -54.307, 126.714, -145.953, 75.908, 171.637]
  MoveL 8602 to (4.76, -20.36, -44.5) mm, rotated rx -180 ry 0 rz 0.01 deg; joints [33.005, -54.25, 126.572, -145.811, 75.86, 171.555]
  MoveC 8603 to (3.66, -18.8, -44.5) mm, rotated rx -180 ry 0 rz 0.01 deg; joints [33.038, -54.191, 126.43, -145.766, 75.797, 171.498] to (1.82, -19.33, -44.5) mm, rotated rx 180 ry 0 rz 0.01 deg; joints [32.971, -54.147, 126.33, -145.826, 75.738, 171.483]
  MoveL 8604 to (0.09, -21.49, -44.5) mm, rotated rx -180 ry 0 rz 0.01 deg; joints [32.843, -54.135, 126.308, -145.954, 75.708, 171.51]
  MoveC 8605 to (-0.12, -22.22, -44.5) mm, rotated rx -180 ry 0 rz 0.01 deg; joints [32.809, -54.142, 126.325, -145.99, 75.711, 171.525] to (0.24, -22.89, -44.5) mm, rotated rx -180 ry 0 rz 0.01 deg; joints [32.792, -54.164, 126.378, -146.012, 75.734, 171.548]
  MoveL 8606 to (7.77, -29, -44.5) mm, rotated rx -180 ry 0 rz 0.01 deg; joints [32.743, -54.486, 127.147, -146.125, 76.096, 171.818]
  MoveL 8607 to (7.66, -30.63, -44.5) mm, rotated rx 180 ry 0 rz 0.01 deg; joints [32.676, -54.511, 127.21, -146.197, 76.117, 171.856]
  MoveL 8608 to (7.44, -30.76, -44.5) mm, rotated rx 180 ry 0 rz 0.01 deg; joints [32.665, -54.507, 127.201, -146.208, 76.111, 171.856]
  MoveL 8609 to (6.62, -31.07, -44.5) mm, rotated rx -180 ry 0 rz 0.01 deg; joints [32.633, -54.488, 127.159, -146.238, 76.086, 171.851]
  MoveL 8610 to (5.41, -31.27, -44.5) mm, rotated rx 180 ry 0 rz 0.01 deg; joints [32.594, -54.457, 127.086, -146.271, 76.045, 171.837]
  MoveL 8611 to (-25.72, -31.27, -44.5) mm, rotated rx -180 ry 0 rz 0.01 deg; joints [31.828, -53.552, 124.975, -146.879, 74.908, 171.355]
  MoveL 8612 to (-19.63, -29.44, -44.5) mm, rotated rx -180 ry 0 rz 0.01 deg; joints [32.047, -53.7, 125.314, -146.684, 75.106, 171.403]
  MoveL 8613 to (-19.19, -29.27, -44.5) mm, rotated rx -180 ry 0 rz 0.01 deg; joints [32.064, -53.71, 125.337, -146.669, 75.119, 171.406]
  MoveL 8614 to (-17.96, -28.71, -44.5) mm, rotated rx 180 ry 0 rz 0.01 deg; joints [32.116, -53.736, 125.396, -146.621, 75.156, 171.41]
  MoveL 8615 to (-17.48, -28.44, -44.5) mm, rotated rx -180 ry 0 rz 0.01 deg; joints [32.138, -53.746, 125.417, -146.6, 75.17, 171.411]
  MoveL 8616 to (-7.67, -21.82, -44.5) mm, rotated rx -180 ry 0 rz 0.01 deg; joints [32.636, -53.917, 125.799, -146.123, 75.431, 171.397]
  MoveL 8617 to (-7.37, -21.6, -44.5) mm, rotated rx 180 ry 0 rz 0.01 deg; joints [32.652, -53.922, 125.809, -146.107, 75.439, 171.396]
  MoveL 8618 to (-6.63, -20.97, -44.5) mm, rotated rx 180 ry 0 rz 0.01 deg; joints [32.695, -53.932, 125.832, -146.066, 75.456, 171.392]
  MoveL 8619 to (-6.18, -20.51, -44.5) mm, rotated rx -180 ry 0 rz 0.01 deg; joints [32.724, -53.937, 125.843, -146.037, 75.466, 171.387]
  MoveL 8620 to (1.7, -10.66, -44.5) mm, rotated rx -180 ry 0 rz 0.01 deg; joints [33.303, -53.991, 125.943, -145.455, 75.606, 171.261]
  MoveL 8621 to (1.99, -10.24, -44.5) mm, rotated rx -180 ry 0 rz 0.01 deg; joints [33.327, -53.992, 125.944, -145.431, 75.61, 171.255]
  MoveL 8622 to (5.98, -3.35, -44.5) mm, rotated rx 180 ry 0 rz 0.01 deg; joints [33.693, -53.983, 125.906, -145.054, 75.651, 171.141]
  MoveL 8623 to (6.19, -2.9, -44.5) mm, rotated rx 180 ry 0 rz 0.01 deg; joints [33.716, -53.981, 125.901, -145.03, 75.652, 171.133]
  MoveL 8624 to (10.27, 7.43, -44.5) mm, rotated rx -180 ry 0 rz 0.01 deg; joints [34.216, -53.911, 125.71, -144.505, 75.644, 170.931]
  MoveL 8625 to (10.27, -25.87, -44.5) mm, rotated rx 180 ry 0 rz 0.01 deg; joints [32.929, -54.503, 127.18, -145.937, 76.14, 171.779]
  MoveL 8626 to (10.22, -26.94, -44.5) mm, rotated rx 180 ry 0 rz 0.01 deg; joints [32.886, -54.52, 127.222, -145.985, 76.154, 171.805]
  MoveL 8627 to (10.02, -27.8, -44.5) mm, rotated rx -180 ry 0 rz 0.01 deg; joints [32.847, -54.529, 127.246, -146.027, 76.16, 171.823]
  MoveL 8628 to (9.68, -28.6, -44.5) mm, rotated rx 180 ry 0 rz 0.01 deg; joints [32.807, -54.533, 127.257, -146.068, 76.159, 171.838]
  MoveL 8629 to (9.37, -28.67, -44.5) mm, rotated rx 180 ry 0 rz 0.01 deg; joints [32.796, -54.526, 127.24, -146.078, 76.149, 171.835]
  MoveL 8630 to (8.67, -28.05, -44.5) mm, rotated rx 180 ry 0 rz 0.01 deg; joints [32.803, -54.495, 127.166, -146.065, 76.115, 171.808]
  MoveL 8631 to (5.05, -25.58, -44.5) mm, rotated rx 180 ry 0 rz 0.01 deg; joints [32.809, -54.349, 126.817, -146.031, 75.948, 171.69]
  MoveL 8632 to (5.31, -26.06, -44.5) mm, rotated rx 180 ry 0 rz 0.01 deg; joints [32.796, -54.365, 126.856, -146.047, 75.964, 171.706]
  MoveL 8633 to (5.26, -25.18, -44.5) mm, rotated rx 180 ry 0 rz 0.01 deg; joints [32.829, -54.348, 126.814, -146.01, 75.949, 171.683]
  MoveL 8634 to (3.74, -18.75, -44.74) mm, rotated rx 180 ry 0 rz 0.01 deg; joints [33.042, -54.176, 126.432, -145.764, 75.811, 171.507]
  MoveL 8635 to (-2.76, -17.57, -44.99) mm, rotated rx 180 ry 0 rz 0.01 deg; joints [32.924, -53.952, 125.943, -145.846, 75.572, 171.384]
  MoveL 8636 to (-6.45, -23.05, -45.23) mm, rotated rx 180 ry 0 rz 0.01 deg; joints [32.62, -53.925, 125.93, -146.157, 75.531, 171.473]
  MoveL 8637 to (-2.92, -28.62, -45.48) mm, rotated rx 180 ry 0 rz 0.01 deg; joints [32.49, -54.107, 126.406, -146.331, 75.754, 171.676]
  MoveL 8638 to (3.61, -27.62, -45.72) mm, rotated rx 180 ry 0 rz 0.01 deg; joints [32.693, -54.26, 126.801, -146.159, 75.988, 171.761]
  MoveL 8639 to (5.31, -21.25, -45.96) mm, rotated rx -180 ry 0 rz 0.01 deg; joints [32.985, -54.182, 126.639, -145.85, 75.967, 171.637]
  MoveL 8640 to (0.16, -17.13, -46.21) mm, rotated rx -180 ry 0 rz 0.01 deg; joints [33.015, -53.947, 126.112, -145.778, 75.732, 171.461]
  MoveL 8641 to (-5.69, -20.19, -46.45) mm, rotated rx -180 ry 0 rz 0.01 deg; joints [32.75, -53.816, 125.85, -146.029, 75.578, 171.455]
  MoveL 8642 to (-5.22, -26.78, -46.7) mm, rotated rx 180 ry 0 rz 0.01 deg; joints [32.506, -53.927, 126.164, -146.306, 75.705, 171.636]
  MoveL 8643 to (1, -29, -46.94) mm, rotated rx 180 ry 0 rz 0.01 deg; joints [32.574, -54.127, 126.677, -146.28, 75.976, 171.797]
  MoveL 8644 to (5.52, -24.19, -47.18) mm, rotated rx 180 ry 0 rz 0.01 deg; joints [32.876, -54.157, 126.772, -145.983, 76.081, 171.757]
  MoveL 8645 to (2.94, -18.12, -47.43) mm, rotated rx -180 ry 0 rz 0.01 deg; joints [33.048, -53.961, 126.334, -145.775, 75.909, 171.573]
  MoveL 8646 to (-3.66, -18.05, -47.67) mm, rotated rx 180 ry 0 rz 0.01 deg; joints [32.885, -53.755, 125.886, -145.906, 75.681, 171.476]
  MoveL 8647 to (-6.38, -24.06, -47.91) mm, rotated rx -180 ry 0 rz 0.01 deg; joints [32.584, -53.765, 125.962, -146.221, 75.684, 171.592]
  MoveL 8648 to (-1.95, -28.96, -48.16) mm, rotated rx 180 ry 0 rz 0.01 deg; joints [32.503, -53.959, 126.469, -146.348, 75.931, 171.792]
  MoveL 8649 to (4.31, -26.88, -48.4) mm, rotated rx 180 ry 0 rz 0.01 deg; joints [32.741, -54.086, 126.799, -146.133, 76.14, 171.848]
  MoveL 8650 to (4.91, -20.31, -48.65) mm, rotated rx 180 ry 0 rz 0.01 deg; joints [33.014, -53.973, 126.554, -145.839, 76.075, 171.702]
  MoveL 8651 to (-0.86, -17.12, -48.89) mm, rotated rx 180 ry 0 rz 0.01 deg; joints [32.992, -53.737, 126.026, -145.82, 75.83, 171.539]
  MoveL 8652 to (-6.11, -21.13, -49.13) mm, rotated rx -180 ry 0 rz 0.01 deg; joints [32.705, -53.64, 125.845, -146.099, 75.712, 171.565]
  MoveL 8653 to (-4.54, -27.54, -49.38) mm, rotated rx -180 ry 0 rz 0.01 deg; joints [32.495, -53.779, 126.226, -146.347, 75.877, 171.759]
  MoveL 8654 to (1.97, -28.67, -49.62) mm, rotated rx 180 ry 0 rz 0.01 deg; joints [32.613, -53.967, 126.711, -146.268, 76.144, 171.898]
  MoveL 8655 to (5.62, -23.17, -49.87) mm, rotated rx -180 ry 0 rz 0.01 deg; joints [32.92, -53.96, 126.717, -145.958, 76.206, 171.828]
  MoveL 8656 to (2.04, -17.62, -50.11) mm, rotated rx -180 ry 0 rz 0.01 deg; joints [33.046, -53.747, 126.235, -145.793, 76.005, 171.641]
  MoveL 8657 to (-4.47, -18.67, -50.35) mm, rotated rx -180 ry 0 rz 0.01 deg; joints [32.842, -53.563, 125.841, -145.97, 75.796, 171.572]
  MoveL 8658 to (-6.13, -25.06, -50.6) mm, rotated rx -180 ry 0 rz 0.01 deg; joints [32.553, -53.609, 126.003, -146.281, 75.843, 171.714]
  MoveL 8659 to (-0.95, -29.14, -50.84) mm, rotated rx -180 ry 0 rz 0.01 deg; joints [32.523, -53.81, 126.527, -146.356, 76.107, 171.906]
  MoveL 8660 to (4.87, -26.03, -51.09) mm, rotated rx 180 ry 0 rz 0.01 deg; joints [32.791, -53.905, 126.783, -146.106, 76.284, 171.93]
  MoveL 8661 to (4.36, -19.45, -51.33) mm, rotated rx -180 ry 0 rz 0.01 deg; joints [33.035, -53.761, 126.462, -145.834, 76.178, 171.766]
  MoveL 8662 to (-1.87, -17.28, -51.57) mm, rotated rx 180 ry 0 rz 0.01 deg; joints [32.962, -53.531, 125.948, -145.868, 75.931, 171.621]
  MoveL 8663 to (-6.36, -22.11, -51.82) mm, rotated rx 180 ry 0 rz 0.01 deg; joints [32.662, -53.47, 125.853, -146.168, 75.852, 171.679]
  MoveL 8664 to (-3.73, -28.17, -52.06) mm, rotated rx 180 ry 0 rz 0.01 deg; joints [32.492, -53.632, 126.289, -146.379, 76.052, 171.88]
  MoveL 8665 to (2.87, -28.19, -52.3) mm, rotated rx 180 ry 0 rz 0.01 deg; joints [32.656, -53.802, 126.733, -146.249, 76.306, 171.994]
  MoveL 8666 to (5.54, -22.16, -52.55) mm, rotated rx 180 ry 0 rz 0.01 deg; joints [32.96, -53.758, 126.65, -145.936, 76.324, 171.895]
  MoveL 8667 to (1.08, -17.29, -52.79) mm, rotated rx 180 ry 0 rz 0.01 deg; joints [33.037, -53.533, 126.138, -145.818, 76.099, 171.711]
  MoveL 8668 to (-5.17, -19.42, -53.04) mm, rotated rx 180 ry 0 rz 0.01 deg; joints [32.798, -53.376, 125.809, -146.037, 75.916, 171.672]
  MoveL 8669 to (-5.73, -25.99, -53.28) mm, rotated rx -180 ry 0 rz 0.01 deg; joints [32.528, -53.456, 126.053, -146.334, 76.008, 171.836]
  MoveL 8670 to (0.07, -29.14, -53.52) mm, rotated rx 180 ry 0 rz 0.01 deg; joints [32.55, -53.657, 126.578, -146.356, 76.281, 172.015]
  MoveL 8671 to (5.29, -25.1, -53.77) mm, rotated rx -180 ry 0 rz 0.01 deg; joints [32.839, -53.719, 126.752, -146.077, 76.421, 172.007]
  MoveL 8672 to (3.67, -18.7, -54.01) mm, rotated rx 180 ry 0 rz 0.01 deg; joints [33.048, -53.548, 126.365, -145.836, 76.277, 171.83]
  MoveL 8673 to (-2.84, -17.61, -54.26) mm, rotated rx -180 ry 0 rz 0.01 deg; joints [32.927, -53.329, 125.879, -145.922, 76.035, 171.707]
  MoveL 8674 to (-6.45, -23.13, -54.5) mm, rotated rx 180 ry 0 rz 0.01 deg; joints [32.623, -53.305, 125.873, -146.234, 75.999, 171.795]
  MoveC 8675 to (-0.84, -28.74, -54.5) mm, rotated rx -180 ry 0 rz 0.01 deg; joints [32.544, -53.558, 126.492, -146.364, 76.29, 172.024] to (4.76, -23.13, -54.5) mm, rotated rx -180 ry 0 rz 0.01 deg; joints [32.904, -53.621, 126.627, -146.009, 76.409, 171.975]
  MoveL 8676 to (4.76, -20.36, -54.5) mm, rotated rx -180 ry 0 rz 0.01 deg; joints [33.011, -53.574, 126.507, -145.889, 76.367, 171.907]
  MoveC 8677 to (3.66, -18.8, -54.5) mm, rotated rx 180 ry 0 rz 0.01 deg; joints [33.044, -53.516, 126.365, -145.845, 76.302, 171.85] to (1.82, -19.33, -54.5) mm, rotated rx -180 ry 0 rz 0.01 deg; joints [32.977, -53.473, 126.265, -145.905, 76.243, 171.833]
  MoveL 8678 to (-0.77, -22.57, -54.5) mm, rotated rx 180 ry 0 rz 0.01 deg; joints [32.786, -53.456, 126.231, -146.096, 76.199, 171.872]
  MoveC 8679 to (-1.01, -24.64, -54.5) mm, rotated rx -180 ry 0 rz 0.01 deg; joints [32.699, -53.484, 126.305, -146.191, 76.222, 171.92] to (0.76, -25.76, -54.5) mm, rotated rx -180 ry 0 rz 0.01 deg; joints [32.7, -53.553, 126.472, -146.203, 76.303, 171.976]
  MoveL 8680 to (2.65, -25.76, -54.5) mm, rotated rx -180 ry 0 rz 0.01 deg; joints [32.748, -53.606, 126.599, -146.165, 76.372, 172.006]
  MoveC 8681 to (4.15, -25.14, -54.5) mm, rotated rx 180 ry 0 rz 0.01 deg; joints [32.81, -53.638, 126.672, -146.108, 76.417, 172.015] to (4.76, -23.64, -54.5) mm, rotated rx -180 ry 0 rz 0.01 deg; joints [32.884, -53.63, 126.649, -146.031, 76.417, 171.988]
  MoveL 8682 to (4.76, -23.13, -54.5) mm, rotated rx -180 ry 0 rz 0.01 deg; joints [32.904, -53.621, 126.627, -146.009, 76.409, 171.975]
  MoveL 8683 to (3.55, -23.4, -54.5) mm, rotated rx -180 ry 0 rz 0.01 deg; joints [32.863, -53.591, 126.557, -146.045, 76.369, 171.963]
  MoveL 8684 to (4.05, -24.46, -54.5) mm, rotated rx 180 ry 0 rz 0.01 deg; joints [32.833, -53.623, 126.636, -146.081, 76.403, 171.997]
  MoveL 8685 to (4.24, -24.7, -54.5) mm, rotated rx 180 ry 0 rz 0.01 deg; joints [32.829, -53.633, 126.66, -146.087, 76.414, 172.006]
  MoveL 8686 to (8.68, -28.03, -54.5) mm, rotated rx 180 ry 0 rz 0.01 deg; joints [32.811, -53.813, 127.1, -146.14, 76.627, 172.16]
  MoveL 8687 to (9.37, -28.67, -54.5) mm, rotated rx -180 ry 0 rz 0.01 deg; joints [32.803, -53.843, 127.174, -146.154, 76.662, 172.187]
  MoveL 8688 to (9.68, -28.6, -54.5) mm, rotated rx 180 ry 0 rz 0.01 deg; joints [32.813, -53.851, 127.192, -146.145, 76.673, 172.19]
  MoveL 8689 to (10.02, -27.8, -54.5) mm, rotated rx 180 ry 0 rz 0.01 deg; joints [32.854, -53.847, 127.181, -146.103, 76.673, 172.176]
  MoveL 8690 to (10.22, -26.94, -54.5) mm, rotated rx 180 ry 0 rz 0.01 deg; joints [32.893, -53.838, 127.156, -146.062, 76.667, 172.158]
  MoveL 8691 to (10.27, -25.87, -54.5) mm, rotated rx 180 ry 0 rz 0.01 deg; joints [32.936, -53.821, 127.114, -146.014, 76.652, 172.132]
  MoveL 8692 to (10.27, 7.41, -54.5) mm, rotated rx 180 ry 0 rz 0.01 deg; joints [34.221, -53.243, 125.647, -144.588, 76.137, 171.291]
  MoveL 8693 to (6.19, -2.9, -54.5) mm, rotated rx -180 ry 0 rz 0.01 deg; joints [33.723, -53.311, 125.836, -145.111, 76.149, 171.489]
  MoveL 8694 to (5.98, -3.35, -54.5) mm, rotated rx 180 ry 0 rz 0.01 deg; joints [33.7, -53.313, 125.841, -145.135, 76.148, 171.497]
  MoveL 8695 to (1.99, -10.24, -54.5) mm, rotated rx -180 ry 0 rz 0.01 deg; joints [33.333, -53.321, 125.879, -145.511, 76.11, 171.607]
  MoveL 8696 to (1.7, -10.66, -54.5) mm, rotated rx 180 ry 0 rz 0.01 deg; joints [33.31, -53.321, 125.878, -145.534, 76.106, 171.613]
  MoveL 8697 to (-6.17, -20.5, -54.5) mm, rotated rx 180 ry 0 rz 0.01 deg; joints [32.732, -53.268, 125.778, -146.115, 75.969, 171.734]
  MoveL 8698 to (-6.63, -20.97, -54.5) mm, rotated rx -180 ry 0 rz 0.01 deg; joints [32.702, -53.263, 125.768, -146.144, 75.96, 171.738]
  MoveL 8699 to (-7.37, -21.6, -54.5) mm, rotated rx 180 ry 0 rz 0.01 deg; joints [32.659, -53.252, 125.745, -146.186, 75.942, 171.742]
  MoveL 8700 to (-7.66, -21.82, -54.5) mm, rotated rx 180 ry 0 rz 0.01 deg; joints [32.643, -53.248, 125.735, -146.201, 75.935, 171.743]
  MoveL 8701 to (-17.25, -28.32, -54.5) mm, rotated rx 180 ry 0 rz 0.01 deg; joints [32.155, -53.085, 125.363, -146.669, 75.68, 171.752]
  MoveL 8702 to (-17.72, -28.59, -54.5) mm, rotated rx -180 ry 0 rz 0.01 deg; joints [32.133, -53.076, 125.343, -146.69, 75.667, 171.751]
  MoveL 8703 to (-19.17, -29.26, -54.5) mm, rotated rx 180 ry 0 rz 0.01 deg; joints [32.071, -53.045, 125.273, -146.747, 75.623, 171.745]
  MoveL 8704 to (-19.62, -29.44, -54.5) mm, rotated rx -180 ry 0 rz 0.01 deg; joints [32.054, -53.035, 125.25, -146.763, 75.609, 171.742]
  MoveL 8705 to (-25.66, -31.27, -54.5) mm, rotated rx -180 ry 0 rz 0.01 deg; joints [31.836, -52.892, 124.915, -146.957, 75.412, 171.691]
  MoveL 8706 to (5.41, -31.27, -54.5) mm, rotated rx 180 ry 0 rz 0.01 deg; joints [32.601, -53.776, 127.02, -146.347, 76.558, 172.187]
  MoveL 8707 to (6.62, -31.07, -54.5) mm, rotated rx -180 ry 0 rz 0.01 deg; joints [32.639, -53.807, 127.093, -146.314, 76.599, 172.201]
  MoveL 8708 to (7.44, -30.76, -54.5) mm, rotated rx 180 ry 0 rz 0.01 deg; joints [32.672, -53.824, 127.135, -146.284, 76.625, 172.207]
  Set speed (500.0 mm/s)
  MoveL 8709 to (7.44, -30.76, 11) mm, rotated rx 180 ry 0 rz 0.01 deg; joints [32.628, -58.229, 127.399, -145.704, 73.184, 169.821]
  Set speed (500.0 mm/s)
  MoveL 8710 to (5.58, -23.91, 11) mm, rotated rx 180 ry 0 rz 0.01 deg; joints [32.85, -58.036, 126.978, -145.438, 73.041, 169.618]
  Set speed (100.0 mm/s)
  MoveL 8711 to (5.58, -23.91, -42.73) mm, rotated rx 180 ry 0 rz 0.01 deg; joints [32.886, -54.455, 126.791, -145.934, 75.851, 171.594]
  MoveL 8712 to (5.6, -23.75, -43.35) mm, rotated rx 180 ry 0 rz 0.01 deg; joints [32.893, -54.41, 126.782, -145.932, 75.881, 171.612]
  MoveL 8713 to (5.63, -23.3, -43.82) mm, rotated rx -180 ry 0 rz 0.01 deg; joints [32.911, -54.372, 126.762, -145.916, 75.899, 171.618]
  MoveL 8714 to (5.61, -22.69, -44) mm, rotated rx -180 ry 0 rz 0.01 deg; joints [32.935, -54.349, 126.733, -145.891, 75.899, 171.609]
  MoveL 8715 to (1.59, -17.45, -44.24) mm, rotated rx 180 ry 0 rz 0.01 deg; joints [33.038, -54.125, 126.234, -145.748, 75.689, 171.423]
  MoveL 8716 to (-4.82, -19.04, -44.49) mm, rotated rx 180 ry 0 rz 0.01 deg; joints [32.815, -53.952, 125.87, -145.946, 75.493, 171.371]
  MoveL 8717 to (-5.94, -25.55, -44.73) mm, rotated rx -180 ry 0 rz 0.01 deg; joints [32.535, -54.016, 126.075, -146.252, 75.561, 171.526]
  MoveL 8718 to (-0.42, -29.18, -44.98) mm, rotated rx 180 ry 0 rz 0.01 deg; joints [32.531, -54.222, 126.601, -146.301, 75.827, 171.711]
  MoveL 8719 to (5.12, -25.58, -45.22) mm, rotated rx -180 ry 0 rz 0.01 deg; joints [32.811, -54.302, 126.817, -146.036, 75.987, 171.716]
  MoveL 8720 to (4.03, -19.06, -45.46) mm, rotated rx 180 ry 0 rz 0.01 deg; joints [33.038, -54.141, 126.461, -145.777, 75.863, 171.545]
  MoveL 8721 to (-2.37, -17.44, -45.71) mm, rotated rx 180 ry 0 rz 0.01 deg; joints [32.939, -53.913, 125.959, -145.838, 75.62, 171.412]
  MoveL 8722 to (-6.42, -22.66, -45.95) mm, rotated rx 180 ry 0 rz 0.01 deg; joints [32.636, -53.871, 125.911, -146.146, 75.562, 171.488]
  MoveL 8723 to (-3.26, -28.46, -46.2) mm, rotated rx -180 ry 0 rz 0.01 deg; joints [32.489, -54.045, 126.372, -146.336, 75.775, 171.691]
  MoveL 8724 to (3.32, -27.89, -46.44) mm, rotated rx 180 ry 0 rz 0.01 deg; joints [32.676, -54.208, 126.789, -146.182, 76.019, 171.789]
  MoveL 8725 to (5.44, -21.64, -46.68) mm, rotated rx 180 ry 0 rz 0.01 deg; joints [32.974, -54.144, 126.659, -145.87, 76.014, 171.675]
  MoveL 8726 to (0.55, -17.19, -46.93) mm, rotated rx -180 ry 0 rz 0.01 deg; joints [33.023, -53.91, 126.137, -145.779, 75.783, 171.494]
  MoveL 8727 to (-5.48, -19.88, -47.17) mm, rotated rx 180 ry 0 rz 0.01 deg; joints [32.768, -53.768, 125.846, -146.017, 75.617, 171.476]
  MoveL 8728 to (-5.43, -26.49, -47.42) mm, rotated rx 180 ry 0 rz 0.01 deg; joints [32.513, -53.867, 126.133, -146.304, 75.729, 171.65]
  MoveL 8729 to (0.64, -29.09, -47.66) mm, rotated rx -180 ry 0 rz 0.01 deg; joints [32.563, -54.069, 126.652, -146.297, 76.002, 171.819]
  MoveL 8730 to (5.46, -24.57, -47.9) mm, rotated rx 180 ry 0 rz 0.01 deg; joints [32.861, -54.112, 126.78, -146.006, 76.121, 171.791]
  MoveL 8731 to (3.25, -18.34, -48.15) mm, rotated rx 180 ry 0 rz 0.01 deg; joints [33.047, -53.925, 126.36, -145.784, 75.96, 171.609]
  MoveL 8732 to (-3.34, -17.88, -48.39) mm, rotated rx 180 ry 0 rz 0.01 deg; joints [32.9, -53.713, 125.896, -145.898, 75.726, 171.501]
  MoveL 8733 to (-6.41, -23.73, -48.64) mm, rotated rx 180 ry 0 rz 0.01 deg; joints [32.597, -53.71, 125.94, -146.213, 75.714, 171.608]
  MoveL 8734 to (-2.28, -28.88, -48.88) mm, rotated rx 180 ry 0 rz 0.01 deg; joints [32.498, -53.9, 126.439, -146.356, 75.954, 171.81]
  MoveL 8735 to (4.1, -27.16, -49.12) mm, rotated rx -180 ry 0 rz 0.01 deg; joints [32.726, -54.035, 126.792, -146.155, 76.173, 171.877]
  MoveL 8736 to (5.08, -20.63, -49.37) mm, rotated rx 180 ry 0 rz 0.01 deg; joints [33.006, -53.935, 126.574, -145.855, 76.122, 171.738]
  MoveL 8737 to (-0.51, -17.11, -49.61) mm, rotated rx 180 ry 0 rz 0.01 deg; joints [33.001, -53.698, 126.045, -145.818, 75.879, 171.57]
  MoveL 8738 to (-5.97, -20.83, -49.86) mm, rotated rx 180 ry 0 rz 0.01 deg; joints [32.721, -53.59, 125.837, -146.089, 75.748, 171.585]
  MoveL 8739 to (-4.76, -27.32, -50.1) mm, rotated rx -180 ry 0 rz 0.01 deg; joints [32.498, -53.72, 126.197, -146.347, 75.902, 171.775]
  MoveL 8740 to (1.67, -28.81, -50.35) mm, rotated rx -180 ry 0 rz 0.01 deg; joints [32.601, -53.912, 126.692, -146.285, 76.172, 171.922]
  MoveL 8741 to (5.62, -23.51, -50.59) mm, rotated rx -180 ry 0 rz 0.01 deg; joints [32.908, -53.917, 126.727, -145.978, 76.248, 171.862]
  MoveL 8742 to (2.34, -17.78, -50.83) mm, rotated rx -180 ry 0 rz 0.01 deg; joints [33.048, -53.709, 126.257, -145.799, 76.054, 171.675]
  MoveL 8743 to (-4.22, -18.48, -51.08) mm, rotated rx 180 ry 0 rz 0.01 deg; joints [32.856, -53.518, 125.845, -145.963, 75.838, 171.596]
  MoveL 8744 to (-6.21, -24.77, -51.32) mm, rotated rx 180 ry 0 rz 0.01 deg; joints [32.562, -53.553, 125.981, -146.276, 75.873, 171.73]
  MoveL 8745 to (-1.24, -29.12, -51.57) mm, rotated rx 180 ry 0 rz 0.01 deg; joints [32.517, -53.752, 126.501, -146.366, 76.132, 171.926]
  MoveL 8746 to (4.73, -26.31, -51.81) mm, rotated rx -180 ry 0 rz 0.01 deg; joints [32.777, -53.857, 126.78, -146.126, 76.32, 171.96]
  MoveL 8747 to (4.55, -19.7, -52.05) mm, rotated rx 180 ry 0 rz 0.01 deg; joints [33.03, -53.722, 126.481, -145.846, 76.225, 171.801]
  MoveL 8748 to (-1.57, -17.23, -52.3) mm, rotated rx 180 ry 0 rz 0.01 deg; joints [32.972, -53.49, 125.961, -145.865, 75.977, 171.649]
  MoveL 8749 to (-6.3, -21.84, -52.54) mm, rotated rx -180 ry 0 rz 0.01 deg; joints [32.675, -53.419, 125.841, -146.16, 75.887, 171.698]
  MoveL 8750 to (-3.96, -28.02, -52.79) mm, rotated rx 180 ry 0 rz 0.01 deg; joints [32.493, -53.574, 126.263, -146.382, 76.078, 171.897]
  MoveL 8751 to (2.64, -28.35, -53.03) mm, rotated rx 180 ry 0 rz 0.01 deg; joints [32.645, -53.749, 126.72, -146.266, 76.337, 172.019]
  MoveL 8752 to (5.59, -22.44, -53.27) mm, rotated rx 180 ry 0 rz 0.01 deg; joints [32.95, -53.716, 126.661, -145.953, 76.366, 171.929]
  MoveL 8753 to (1.35, -17.38, -53.52) mm, rotated rx 180 ry 0 rz 0.01 deg; joints [33.041, -53.493, 126.155, -145.822, 76.147, 171.743]
  MoveL 8754 to (-4.99, -19.22, -53.76) mm, rotated rx 180 ry 0 rz 0.01 deg; joints [32.81, -53.329, 125.808, -146.031, 75.956, 171.695]
  MoveL 8755 to (-5.84, -25.77, -54.01) mm, rotated rx 180 ry 0 rz 0.01 deg; joints [32.535, -53.4, 126.031, -146.332, 76.037, 171.854]
  MoveL 8756 to (-0.18, -29.17, -54.25) mm, rotated rx -180 ry 0 rz 0.01 deg; joints [32.543, -53.601, 126.557, -146.368, 76.309, 172.037]
  MoveL 8757 to (5.21, -25.35, -54.49) mm, rotated rx 180 ry 0 rz 0.01 deg; joints [32.828, -53.671, 126.753, -146.095, 76.459, 172.037]
  MoveL 8758 to (3.87, -18.89, -54.74) mm, rotated rx -180 ry 0 rz 0.01 deg; joints [33.046, -53.507, 126.381, -145.846, 76.323, 171.863]
  MoveL 8759 to (-2.6, -17.53, -54.98) mm, rotated rx 180 ry 0 rz 0.01 deg; joints [32.936, -53.286, 125.886, -145.92, 76.079, 171.734]
  MoveL 8760 to (-6.43, -22.9, -55.23) mm, rotated rx -180 ry 0 rz 0.01 deg; joints [32.632, -53.252, 125.859, -146.229, 76.033, 171.815]
  MoveL 8761 to (-3.04, -28.57, -55.47) mm, rotated rx -180 ry 0 rz 0.01 deg; joints [32.496, -53.428, 126.33, -146.408, 76.256, 172.018]
  MoveL 8762 to (3.51, -27.74, -55.71) mm, rotated rx -180 ry 0 rz 0.01 deg; joints [32.693, -53.581, 126.733, -146.242, 76.496, 172.111]
  MoveL 8763 to (5.37, -21.4, -55.96) mm, rotated rx 180 ry 0 rz 0.01 deg; joints [32.987, -53.509, 126.582, -145.933, 76.478, 171.993]
  MoveL 8764 to (0.31, -17.16, -56.2) mm, rotated rx 180 ry 0 rz 0.01 deg; joints [33.025, -53.279, 126.057, -145.855, 76.24, 171.814]
  MoveL 8765 to (-5.61, -20.09, -56.45) mm, rotated rx 180 ry 0 rz 0.01 deg; joints [32.763, -53.146, 125.785, -146.101, 76.081, 171.8]
  MoveL 8766 to (-5.29, -26.69, -56.69) mm, rotated rx -180 ry 0 rz 0.01 deg; joints [32.514, -53.25, 126.089, -146.381, 76.206, 171.977]
  MoveL 8767 to (0.88, -29.04, -56.93) mm, rotated rx 180 ry 0 rz 0.01 deg; joints [32.577, -53.446, 126.604, -146.361, 76.482, 172.143]
  MoveL 8768 to (5.51, -24.33, -57.18) mm, rotated rx 180 ry 0 rz 0.01 deg; joints [32.877, -53.48, 126.71, -146.065, 76.59, 172.11]
  MoveL 8769 to (3.05, -18.2, -57.42) mm, rotated rx 180 ry 0 rz 0.01 deg; joints [33.054, -53.291, 126.278, -145.853, 76.418, 171.927]
  MoveL 8770 to (-3.55, -18, -57.67) mm, rotated rx 180 ry 0 rz 0.01 deg; joints [32.896, -53.086, 125.824, -145.98, 76.185, 171.823]
  MoveL 8771 to (-6.38, -23.97, -57.91) mm, rotated rx -180 ry 0 rz 0.01 deg; joints [32.594, -53.091, 125.889, -146.295, 76.186, 171.934]
  MoveL 8772 to (-2.05, -28.95, -58.15) mm, rotated rx 180 ry 0 rz 0.01 deg; joints [32.508, -53.28, 126.394, -146.425, 76.434, 172.136]
  MoveL 8773 to (4.26, -26.98, -58.4) mm, rotated rx 180 ry 0 rz 0.01 deg; joints [32.743, -53.406, 126.731, -146.214, 76.648, 172.198]
  MoveL 8774 to (4.97, -20.41, -58.64) mm, rotated rx 180 ry 0 rz 0.01 deg; joints [33.018, -53.299, 126.494, -145.918, 76.584, 172.055]
  MoveL 8775 to (-0.76, -17.12, -58.89) mm, rotated rx 180 ry 0 rz 0.01 deg; joints [33.001, -53.068, 125.965, -145.895, 76.335, 171.888]
  MoveL 8776 to (-6.06, -21.05, -59.13) mm, rotated rx 180 ry 0 rz 0.01 deg; joints [32.716, -52.969, 125.776, -146.172, 76.213, 171.908]
  MoveL 8777 to (-4.59, -27.49, -59.38) mm, rotated rx -180 ry 0 rz 0.01 deg; joints [32.502, -53.102, 126.151, -146.422, 76.38, 172.1]
  MoveL 8778 to (1.9, -28.72, -59.62) mm, rotated rx 180 ry 0 rz 0.01 deg; joints [32.616, -53.287, 126.639, -146.346, 76.65, 172.244]
  MoveL 8779 to (5.63, -23.27, -59.86) mm, rotated rx 180 ry 0 rz 0.01 deg; joints [32.924, -53.282, 126.652, -146.037, 76.714, 172.179]
  MoveL 8780 to (2.12, -17.67, -60.11) mm, rotated rx -180 ry 0 rz 0.01 deg; joints [33.053, -53.075, 126.173, -145.869, 76.51, 171.991]
  MoveL 8781 to (-4.41, -18.63, -60.35) mm, rotated rx 180 ry 0 rz 0.01 deg; joints [32.852, -52.892, 125.774, -146.044, 76.297, 171.917]
  MoveL 8782 to (-6.14, -25.01, -60.6) mm, rotated rx -180 ry 0 rz 0.01 deg; joints [32.561, -52.934, 125.93, -146.355, 76.345, 172.055]
  MoveL 8783 to (-1, -29.15, -60.84) mm, rotated rx 180 ry 0 rz 0.01 deg; joints [32.528, -53.13, 126.453, -146.432, 76.612, 172.249]
  MoveL 8784 to (4.86, -26.1, -61.08) mm, rotated rx -180 ry 0 rz 0.01 deg; joints [32.794, -53.225, 126.713, -146.183, 76.792, 172.279]
  MoveL 8785 to (4.41, -19.51, -61.33) mm, rotated rx -180 ry 0 rz 0.01 deg; joints [33.04, -53.086, 126.396, -145.911, 76.683, 172.117]
  MoveL 8786 to (-1.81, -17.28, -61.57) mm, rotated rx 180 ry 0 rz 0.01 deg; joints [32.97, -52.86, 125.881, -145.943, 76.432, 171.967]
  MoveL 8787 to (-6.34, -22.08, -61.82) mm, rotated rx -180 ry 0 rz 0.01 deg; joints [32.671, -52.798, 125.782, -146.242, 76.353, 172.021]
  MoveL 8788 to (-3.76, -28.16, -62.06) mm, rotated rx 180 ry 0 rz 0.01 deg; joints [32.499, -52.954, 126.215, -146.454, 76.556, 172.222]
  MoveL 8789 to (2.85, -28.23, -62.3) mm, rotated rx 180 ry 0 rz 0.01 deg; joints [32.661, -53.122, 126.661, -146.325, 76.813, 172.34]
  MoveL 8790 to (5.55, -22.2, -62.55) mm, rotated rx -180 ry 0 rz 0.01 deg; joints [32.965, -53.08, 126.581, -146.012, 76.829, 172.245]
  MoveL 8791 to (1.12, -17.31, -62.79) mm, rotated rx 180 ry 0 rz 0.01 deg; joints [33.044, -52.859, 126.069, -145.894, 76.601, 172.058]
  MoveL 8792 to (-5.14, -19.41, -63.04) mm, rotated rx -180 ry 0 rz 0.01 deg; joints [32.805, -52.704, 125.738, -146.112, 76.416, 172.016]
  MoveL 8793 to (-5.73, -25.99, -63.28) mm, rotated rx 180 ry 0 rz 0.01 deg; joints [32.535, -52.781, 125.98, -146.408, 76.51, 172.177]
  MoveL 8794 to (0.07, -29.16, -63.52) mm, rotated rx -180 ry 0 rz 0.01 deg; joints [32.556, -52.977, 126.505, -146.43, 76.787, 172.359]
  MoveL 8795 to (5.29, -25.12, -63.77) mm, rotated rx -180 ry 0 rz 0.01 deg; joints [32.845, -53.038, 126.68, -146.152, 76.928, 172.354]
  MoveL 8796 to (3.69, -18.72, -64.01) mm, rotated rx -180 ry 0 rz 0.01 deg; joints [33.055, -52.871, 126.293, -145.911, 76.779, 172.178]
  MoveL 8797 to (-2.82, -17.62, -64.26) mm, rotated rx 180 ry 0 rz 0.01 deg; joints [32.933, -52.656, 125.807, -145.998, 76.534, 172.051]
  MoveL 8798 to (-6.44, -23.15, -64.5) mm, rotated rx -180 ry 0 rz 0.01 deg; joints [32.629, -52.632, 125.801, -146.309, 76.5, 172.137]
  MoveC 8799 to (-0.83, -28.75, -64.5) mm, rotated rx -180 ry 0 rz 0.01 deg; joints [32.55, -52.879, 126.419, -146.438, 76.796, 172.367] to (4.77, -23.15, -64.5) mm, rotated rx 180 ry 0 rz 0.01 deg; joints [32.91, -52.941, 126.554, -146.083, 76.914, 172.322]
  MoveL 8800 to (4.77, -20.36, -64.5) mm, rotated rx -180 ry 0 rz 0.01 deg; joints [33.018, -52.895, 126.434, -145.963, 76.869, 172.254]
  MoveC 8801 to (3.67, -18.8, -64.5) mm, rotated rx -180 ry 0 rz 0.01 deg; joints [33.051, -52.838, 126.292, -145.919, 76.804, 172.197] to (1.83, -19.34, -64.5) mm, rotated rx -180 ry 0 rz 0.01 deg; joints [32.984, -52.797, 126.192, -145.979, 76.745, 172.179]
  MoveL 8802 to (-0.75, -22.59, -64.5) mm, rotated rx 180 ry 0 rz 0.01 deg; joints [32.793, -52.78, 126.16, -146.171, 76.701, 172.217]
  MoveC 8803 to (-0.98, -24.66, -64.5) mm, rotated rx 180 ry 0 rz 0.01 deg; joints [32.706, -52.808, 126.233, -146.265, 76.726, 172.264] to (0.79, -25.76, -64.5) mm, rotated rx 180 ry 0 rz 0.01 deg; joints [32.707, -52.875, 126.4, -146.276, 76.808, 172.321]
  MoveL 8804 to (2.66, -25.76, -64.5) mm, rotated rx -180 ry 0 rz 0.01 deg; joints [32.754, -52.926, 126.525, -146.238, 76.878, 172.352]
  MoveC 8805 to (4.15, -25.15, -64.5) mm, rotated rx 180 ry 0 rz 0.01 deg; joints [32.816, -52.957, 126.599, -146.181, 76.923, 172.361] to (4.77, -23.65, -64.5) mm, rotated rx -180 ry 0 rz 0.01 deg; joints [32.89, -52.949, 126.576, -146.104, 76.922, 172.335]
  MoveL 8806 to (4.77, -23.15, -64.5) mm, rotated rx 180 ry 0 rz 0.01 deg; joints [32.91, -52.941, 126.554, -146.083, 76.914, 172.322]
  MoveL 8807 to (3.56, -23.41, -64.5) mm, rotated rx 180 ry 0 rz 0.01 deg; joints [32.869, -52.912, 126.485, -146.119, 76.873, 172.309]
  MoveL 8808 to (4.06, -24.47, -64.5) mm, rotated rx 180 ry 0 rz 0.01 deg; joints [32.84, -52.943, 126.563, -146.154, 76.908, 172.343]
  MoveL 8809 to (4.25, -24.71, -64.5) mm, rotated rx -180 ry 0 rz 0.01 deg; joints [32.835, -52.953, 126.587, -146.161, 76.919, 172.352]
  MoveL 8810 to (8.68, -28.03, -64.5) mm, rotated rx 180 ry 0 rz 0.01 deg; joints [32.818, -53.128, 127.026, -146.213, 77.136, 172.507]
  MoveL 8811 to (9.37, -28.67, -64.5) mm, rotated rx -180 ry 0 rz 0.01 deg; joints [32.81, -53.157, 127.099, -146.226, 77.171, 172.534]
  MoveL 8812 to (9.68, -28.6, -64.5) mm, rotated rx -180 ry 0 rz 0.01 deg; joints [32.82, -53.165, 127.117, -146.217, 77.181, 172.538]
  MoveL 8813 to (10.02, -27.8, -64.5) mm, rotated rx -180 ry 0 rz 0.01 deg; joints [32.86, -53.161, 127.106, -146.175, 77.181, 172.524]
  MoveL 8814 to (10.22, -26.94, -64.5) mm, rotated rx 180 ry 0 rz 0.01 deg; joints [32.899, -53.152, 127.082, -146.134, 77.175, 172.506]
  MoveL 8815 to (10.27, -25.87, -64.5) mm, rotated rx -180 ry 0 rz 0.01 deg; joints [32.943, -53.136, 127.039, -146.086, 77.16, 172.481]
  MoveL 8816 to (10.27, 7.39, -64.5) mm, rotated rx 180 ry 0 rz 0.01 deg; joints [34.227, -52.572, 125.574, -144.666, 76.626, 171.646]
  MoveL 8817 to (6.19, -2.9, -64.5) mm, rotated rx -180 ry 0 rz 0.01 deg; joints [33.729, -52.638, 125.762, -145.187, 76.642, 171.84]
  MoveL 8818 to (5.98, -3.35, -64.5) mm, rotated rx 180 ry 0 rz 0.01 deg; joints [33.706, -52.64, 125.768, -145.211, 76.642, 171.848]
  MoveL 8819 to (1.99, -10.24, -64.5) mm, rotated rx 180 ry 0 rz 0.01 deg; joints [33.34, -52.648, 125.805, -145.586, 76.606, 171.955]
  MoveL 8820 to (1.71, -10.65, -64.5) mm, rotated rx 180 ry 0 rz 0.01 deg; joints [33.317, -52.647, 125.805, -145.61, 76.602, 171.961]
  MoveL 8821 to (-5.9, -20.24, -64.5) mm, rotated rx -180 ry 0 rz 0.01 deg; joints [32.755, -52.598, 125.711, -146.174, 76.474, 172.074]
  MoveL 8822 to (-6.32, -20.67, -64.5) mm, rotated rx -180 ry 0 rz 0.01 deg; joints [32.728, -52.594, 125.702, -146.201, 76.465, 172.078]
  MoveL 8823 to (-7.32, -21.56, -64.5) mm, rotated rx 180 ry 0 rz 0.01 deg; joints [32.669, -52.581, 125.672, -146.259, 76.442, 172.083]
  MoveL 8824 to (-7.66, -21.82, -64.5) mm, rotated rx 180 ry 0 rz 0.01 deg; joints [32.65, -52.576, 125.661, -146.276, 76.434, 172.084]
  MoveL 8825 to (-17.25, -28.33, -64.5) mm, rotated rx 180 ry 0 rz 0.01 deg; joints [32.161, -52.416, 125.29, -146.745, 76.179, 172.087]
  MoveL 8826 to (-17.74, -28.61, -64.5) mm, rotated rx -180 ry 0 rz 0.01 deg; joints [32.138, -52.407, 125.269, -146.766, 76.165, 172.086]
  MoveL 8827 to (-19.19, -29.27, -64.5) mm, rotated rx -180 ry 0 rz 0.01 deg; joints [32.077, -52.377, 125.199, -146.823, 76.121, 172.079]
  MoveL 8828 to (-19.61, -29.44, -64.5) mm, rotated rx 180 ry 0 rz 0.01 deg; joints [32.06, -52.367, 125.176, -146.838, 76.108, 172.076]
  MoveL 8829 to (-25.63, -31.27, -64.5) mm, rotated rx 180 ry 0 rz 0.01 deg; joints [31.844, -52.228, 124.843, -147.032, 75.911, 172.023]
  MoveL 8830 to (5.41, -31.27, -64.5) mm, rotated rx 180 ry 0 rz 0.01 deg; joints [32.608, -53.092, 126.946, -146.42, 77.067, 172.532]
  MoveL 8831 to (6.62, -31.07, -64.5) mm, rotated rx 180 ry 0 rz 0.01 deg; joints [32.646, -53.122, 127.019, -146.386, 77.109, 172.547]
  Set speed (500.0 mm/s)
  MoveL 8832 to (6.62, -31.07, 11.77) mm, rotated rx -180 ry 0 rz 0.01 deg; joints [32.595, -58.259, 127.358, -145.726, 73.118, 169.789]
  Set speed (500.0 mm/s)
  MoveL 8833 to (-399.07, -22.36, 11.77) mm, rotated rx -180 ry 0 rz 0.01 deg; joints [24.941, -42.811, 95.517, -149.899, 57.269, 163.688]
  Set speed (100.0 mm/s)
  MoveL 8834 to (-399.09, -22.53, 11.15) mm, rotated rx -180 ry 0 rz 0.01 deg; joints [24.936, -42.784, 95.522, -149.915, 57.294, 163.71]
  MoveL 8835 to (-399.11, -22.97, 10.68) mm, rotated rx 180 ry 0 rz 0.01 deg; joints [24.921, -42.77, 95.537, -149.941, 57.316, 163.737]
  MoveL 8836 to (-399.1, -23.59, 10.5) mm, rotated rx -180 ry 0 rz 0.01 deg; joints [24.901, -42.774, 95.565, -149.971, 57.33, 163.763]
  MoveL 8837 to (-395.07, -28.82, 10.26) mm, rotated rx 180 ry 0 rz 0.01 deg; joints [24.791, -43.045, 96.15, -150.196, 57.569, 164.018]
  MoveL 8838 to (-388.66, -27.23, 10.01) mm, rotated rx 180 ry 0 rz 0.01 deg; joints [24.941, -43.285, 96.662, -150.112, 57.85, 164.085]
  MoveL 8839 to (-387.55, -20.72, 9.77) mm, rotated rx 180 ry 0 rz 0.01 deg; joints [25.173, -43.195, 96.488, -149.824, 57.847, 163.895]
  MoveL 8840 to (-393.07, -17.1, 9.52) mm, rotated rx 180 ry 0 rz 0.01 deg; joints [25.207, -42.867, 95.836, -149.682, 57.576, 163.68]
  MoveL 8841 to (-398.61, -20.7, 9.28) mm, rotated rx 180 ry 0 rz 0.01 deg; joints [25.004, -42.682, 95.486, -149.859, 57.373, 163.707]
  MoveL 8842 to (-397.52, -27.21, 9.04) mm, rotated rx -180 ry 0 rz 0.01 deg; joints [24.807, -42.847, 95.859, -150.148, 57.493, 163.953]
  MoveL 8843 to (-391.12, -28.83, 8.79) mm, rotated rx -180 ry 0 rz 0.01 deg; joints [24.852, -43.15, 96.506, -150.206, 57.805, 164.128]
  MoveL 8844 to (-387.07, -23.62, 8.55) mm, rotated rx -180 ry 0 rz 0.01 deg; joints [25.086, -43.215, 96.652, -149.967, 57.945, 164.033]
  MoveL 8845 to (-390.23, -17.81, 8.3) mm, rotated rx -180 ry 0 rz 0.01 deg; joints [25.228, -42.95, 96.122, -149.724, 57.758, 163.789]
  MoveL 8846 to (-396.81, -18.38, 8.06) mm, rotated rx 180 ry 0 rz 0.01 deg; joints [25.108, -42.659, 95.55, -149.769, 57.48, 163.695]
  MoveL 8847 to (-398.92, -24.64, 7.82) mm, rotated rx -180 ry 0 rz 0.01 deg; joints [24.871, -42.677, 95.622, -150.054, 57.455, 163.874]
  MoveL 8848 to (-394.04, -29.08, 7.57) mm, rotated rx -180 ry 0 rz 0.01 deg; joints [24.799, -42.969, 96.251, -150.242, 57.726, 164.117]
  MoveL 8849 to (-388.01, -26.39, 7.33) mm, rotated rx -180 ry 0 rz 0.01 deg; joints [24.981, -43.17, 96.682, -150.109, 57.979, 164.141]
  MoveL 8850 to (-388.06, -19.79, 7.08) mm, rotated rx -180 ry 0 rz 0.01 deg; joints [25.197, -43.027, 96.399, -149.821, 57.923, 163.927]
  MoveL 8851 to (-394.13, -17.19, 6.84) mm, rotated rx 180 ry 0 rz 0.01 deg; joints [25.189, -42.696, 95.74, -149.727, 57.636, 163.736]
  MoveL 8852 to (-398.95, -21.71, 6.6) mm, rotated rx 180 ry 0 rz 0.01 deg; joints [24.968, -42.561, 95.494, -149.942, 57.474, 163.807]
  MoveL 8853 to (-396.73, -27.93, 6.35) mm, rotated rx 180 ry 0 rz 0.01 deg; joints [24.797, -42.77, 95.957, -150.215, 57.643, 164.062]
  MoveL 8854 to (-390.15, -28.4, 6.11) mm, rotated rx 180 ry 0 rz 0.01 deg; joints [24.882, -43.058, 96.572, -150.221, 57.952, 164.202]
  MoveL 8855 to (-387.08, -22.55, 5.86) mm, rotated rx 180 ry 0 rz 0.01 deg; joints [25.123, -43.066, 96.602, -149.957, 58.042, 164.069]
  MoveL 8856 to (-391.21, -17.39, 5.62) mm, rotated rx -180 ry 0 rz 0.01 deg; joints [25.228, -42.771, 96.012, -149.745, 57.818, 163.829]
  MoveL 8857 to (-397.59, -19.11, 5.37) mm, rotated rx -180 ry 0 rz 0.01 deg; joints [25.074, -42.512, 95.506, -149.841, 57.558, 163.777]
  MoveL 8858 to (-398.57, -25.64, 5.13) mm, rotated rx -180 ry 0 rz 0.01 deg; joints [24.845, -42.586, 95.693, -150.135, 57.587, 163.985]
  MoveL 8859 to (-392.98, -29.16, 4.89) mm, rotated rx -180 ry 0 rz 0.01 deg; joints [24.815, -42.89, 96.347, -150.279, 57.882, 164.209]
  MoveL 8860 to (-387.52, -25.45, 4.64) mm, rotated rx 180 ry 0 rz 0.01 deg; joints [25.021, -43.046, 96.683, -150.103, 58.099, 164.19]
  MoveL 8861 to (-388.73, -18.96, 4.4) mm, rotated rx -180 ry 0 rz 0.01 deg; joints [25.216, -42.854, 96.3, -149.824, 57.992, 163.959]
  MoveL 8862 to (-395.16, -17.47, 4.15) mm, rotated rx -180 ry 0 rz 0.01 deg; joints [25.166, -42.529, 95.655, -149.779, 57.699, 163.799]
  MoveL 8863 to (-399.11, -22.76, 3.91) mm, rotated rx 180 ry 0 rz 0.01 deg; joints [24.932, -42.448, 95.521, -150.026, 57.584, 163.911]
  MoveL 8864 to (-395.83, -28.5, 3.67) mm, rotated rx 180 ry 0 rz 0.01 deg; joints [24.794, -42.694, 96.059, -150.274, 57.796, 164.169]
  MoveL 8865 to (-389.26, -27.8, 3.42) mm, rotated rx -180 ry 0 rz 0.01 deg; joints [24.917, -42.957, 96.622, -150.228, 58.093, 164.269]
  MoveL 8866 to (-387.28, -21.5, 3.18) mm, rotated rx 180 ry 0 rz 0.01 deg; joints [25.156, -42.91, 96.537, -149.948, 58.13, 164.103]
  MoveL 8867 to (-392.25, -17.15, 2.93) mm, rotated rx -180 ry 0 rz 0.01 deg; joints [25.222, -42.594, 95.903, -149.774, 57.875, 163.874]
  MoveL 8868 to (-398.22, -19.97, 2.69) mm, rotated rx -180 ry 0 rz 0.01 deg; joints [25.038, -42.375, 95.481, -149.917, 57.644, 163.866]
  MoveL 8869 to (-398.04, -26.57, 2.45) mm, rotated rx -180 ry 0 rz 0.01 deg; joints [24.825, -42.501, 95.776, -150.211, 57.727, 164.097]
  MoveL 8870 to (-391.92, -29.05, 2.2) mm, rotated rx -180 ry 0 rz 0.01 deg; joints [24.836, -42.807, 96.434, -150.307, 58.035, 164.296]
  MoveL 8871 to (-387.19, -24.43, 1.96) mm, rotated rx -180 ry 0 rz 0.01 deg; joints [25.061, -42.913, 96.665, -150.093, 58.211, 164.234]
  MoveL 8872 to (-389.53, -18.25, 1.71) mm, rotated rx -180 ry 0 rz 0.01 deg; joints [25.228, -42.677, 96.193, -149.832, 58.056, 163.993]
  MoveL 8873 to (-396.13, -17.92, 1.47) mm, rotated rx -180 ry 0 rz 0.01 deg; joints [25.138, -42.369, 95.582, -149.838, 57.767, 163.868]
  MoveL 8874 to (-399.08, -23.83, 1.23) mm, rotated rx 180 ry 0 rz 0.01 deg; joints [24.9, -42.344, 95.564, -150.109, 57.702, 164.019]
  MoveL 8875 to (-394.84, -28.9, 0.98) mm, rotated rx 180 ry 0 rz 0.01 deg; joints [24.798, -42.618, 96.161, -150.325, 57.951, 164.27]
  MoveL 8876 to (-388.5, -27.05, 0.74) mm, rotated rx -180 ry 0 rz 0.01 deg; joints [24.955, -42.848, 96.655, -150.229, 58.227, 164.329]
  MoveL 8877 to (-387.65, -20.5, 0.49) mm, rotated rx 180 ry 0 rz 0.01 deg; joints [25.184, -42.746, 96.456, -149.942, 58.211, 164.134]
  MoveL 8878 to (-393.31, -17.1, 0.25) mm, rotated rx -180 ry 0 rz 0.01 deg; joints [25.209, -42.419, 95.8, -149.811, 57.933, 163.925]
  MoveL 8879 to (-398.7, -20.92, 0.01) mm, rotated rx 180 ry 0 rz 0.01 deg; joints [25.001, -42.246, 95.473, -149.997, 57.738, 163.961]
  MoveL 8880 to (-397.35, -27.39, -0.24) mm, rotated rx -180 ry 0 rz 0.01 deg; joints [24.81, -42.42, 95.867, -150.282, 57.872, 164.207]
  MoveL 8881 to (-390.89, -28.75, -0.48) mm, rotated rx -180 ry 0 rz 0.01 deg; joints [24.864, -42.719, 96.509, -150.327, 58.186, 164.375]
  MoveL 8882 to (-387.06, -23.37, -0.73) mm, rotated rx 180 ry 0 rz 0.01 deg; joints [25.1, -42.77, 96.628, -150.082, 58.314, 164.272]
  MoveL 8883 to (-390.45, -17.7, -0.97) mm, rotated rx 180 ry 0 rz 0.01 deg; joints [25.234, -42.499, 96.083, -149.847, 58.116, 164.03]
  MoveL 8884 to (-397, -18.54, -1.21) mm, rotated rx 180 ry 0 rz 0.01 deg; joints [25.106, -42.216, 95.524, -149.904, 57.84, 163.944]
  MoveL 8885 to (-398.86, -24.87, -1.46) mm, rotated rx -180 ry 0 rz 0.01 deg; joints [24.87, -42.247, 95.623, -150.191, 57.828, 164.128]
  MoveL 8886 to (-393.8, -29.12, -1.7) mm, rotated rx -180 ry 0 rz 0.01 deg; joints [24.808, -42.54, 96.259, -150.368, 58.107, 164.367]
  MoveL 8887 to (-387.88, -26.18, -1.95) mm, rotated rx -180 ry 0 rz 0.01 deg; joints [24.995, -42.73, 96.67, -150.225, 58.354, 164.382]
  MoveL 8888 to (-388.2, -19.59, -2.19) mm, rotated rx 180 ry 0 rz 0.01 deg; joints [25.208, -42.576, 96.362, -149.939, 58.284, 164.165]
  MoveL 8889 to (-394.37, -17.24, -2.43) mm, rotated rx 180 ry 0 rz 0.01 deg; joints [25.19, -42.248, 95.704, -149.857, 57.993, 163.981]
  MoveL 8890 to (-399, -21.95, -2.68) mm, rotated rx 180 ry 0 rz 0.01 deg; joints [24.965, -42.126, 95.484, -150.079, 57.841, 164.06]
  MoveL 8891 to (-396.54, -28.07, -2.92) mm, rotated rx 180 ry 0 rz 0.01 deg; joints [24.801, -42.342, 95.965, -150.346, 58.022, 164.315]
  MoveL 8892 to (-389.94, -28.27, -3.17) mm, rotated rx -180 ry 0 rz 0.01 deg; joints [24.896, -42.623, 96.57, -150.339, 58.331, 164.446]
  MoveL 8893 to (-387.11, -22.31, -3.41) mm, rotated rx 180 ry 0 rz 0.01 deg; joints [25.136, -42.619, 96.573, -150.072, 58.408, 164.307]
  MoveL 8894 to (-391.44, -17.32, -3.65) mm, rotated rx -180 ry 0 rz 0.01 deg; joints [25.233, -42.32, 95.971, -149.869, 58.174, 164.07]
  MoveL 8895 to (-397.74, -19.3, -3.9) mm, rotated rx -180 ry 0 rz 0.01 deg; joints [25.071, -42.071, 95.483, -149.976, 57.919, 164.027]
  MoveL 8896 to (-398.46, -25.86, -4.14) mm, rotated rx 180 ry 0 rz 0.01 deg; joints [24.846, -42.156, 95.695, -150.27, 57.962, 164.239]
  MoveL 8897 to (-392.73, -29.15, -4.39) mm, rotated rx 180 ry 0 rz 0.01 deg; joints [24.825, -42.46, 96.351, -150.402, 58.263, 164.457]
  MoveL 8898 to (-387.43, -25.22, -4.63) mm, rotated rx 180 ry 0 rz 0.01 deg; joints [25.036, -42.603, 96.664, -150.217, 58.472, 164.429]
  MoveL 8899 to (-388.9, -18.78, -4.87) mm, rotated rx -180 ry 0 rz 0.01 deg; joints [25.225, -42.402, 96.259, -149.942, 58.351, 164.197]
  MoveL 8900 to (-395.39, -17.55, -5.12) mm, rotated rx -180 ry 0 rz 0.01 deg; joints [25.165, -42.082, 95.62, -149.909, 58.056, 164.044]
  MoveL 8901 to (-399.12, -23.01, -5.36) mm, rotated rx 180 ry 0 rz 0.01 deg; joints [24.93, -42.014, 95.512, -150.162, 57.952, 164.164]
  MoveL 8902 to (-395.61, -28.61, -5.61) mm, rotated rx -180 ry 0 rz 0.01 deg; joints [24.8, -42.265, 96.065, -150.402, 58.176, 164.419]
  MoveL 8903 to (-389.08, -27.64, -5.85) mm, rotated rx 180 ry 0 rz 0.01 deg; joints [24.931, -42.52, 96.614, -150.344, 58.47, 164.511]
  MoveL 8904 to (-387.35, -21.27, -6.1) mm, rotated rx -180 ry 0 rz 0.01 deg; joints [25.168, -42.46, 96.502, -150.062, 58.494, 164.339]
  MoveL 8905 to (-392.49, -17.13, -6.34) mm, rotated rx -180 ry 0 rz 0.01 deg; joints [25.225, -42.143, 95.861, -149.899, 58.23, 164.115]
  MoveL 8906 to (-398.35, -20.18, -6.58) mm, rotated rx 180 ry 0 rz 0.01 deg; joints [25.035, -41.934, 95.459, -150.052, 58.006, 164.116]
  MoveL 8907 to (-397.9, -26.77, -6.83) mm, rotated rx -180 ry 0 rz 0.01 deg; joints [24.826, -42.071, 95.778, -150.344, 58.102, 164.349]
  MoveL 8908 to (-391.68, -28.99, -7.07) mm, rotated rx 180 ry 0 rz 0.01 deg; joints [24.848, -42.374, 96.434, -150.427, 58.415, 164.541]
  MoveL 8909 to (-387.15, -24.19, -7.32) mm, rotated rx -180 ry 0 rz 0.01 deg; joints [25.076, -42.467, 96.64, -150.206, 58.58, 164.471]
  MoveL 8910 to (-389.73, -18.11, -7.56) mm, rotated rx -180 ry 0 rz 0.01 deg; joints [25.236, -42.224, 96.15, -149.951, 58.413, 164.23]
  MoveL 8911 to (-396.34, -18.05, -7.8) mm, rotated rx 180 ry 0 rz 0.01 deg; joints [25.136, -41.923, 95.549, -149.97, 58.124, 164.114]
  MoveL 8912 to (-399.04, -24.07, -8.05) mm, rotated rx 180 ry 0 rz 0.01 deg; joints [24.898, -41.91, 95.557, -150.244, 58.071, 164.27]
  MoveL 8913 to (-394.61, -28.97, -8.29) mm, rotated rx -180 ry 0 rz 0.01 deg; joints [24.805, -42.187, 96.164, -150.451, 58.331, 164.519]
  MoveL 8914 to (-388.35, -26.86, -8.54) mm, rotated rx 180 ry 0 rz 0.01 deg; joints [24.97, -42.408, 96.641, -150.343, 58.602, 164.569]
  MoveL 8915 to (-387.76, -20.29, -8.78) mm, rotated rx -180 ry 0 rz 0.01 deg; joints [25.196, -42.294, 96.416, -150.056, 58.571, 164.37]
  MoveL 8916 to (-393.56, -17.11, -9.02) mm, rotated rx 180 ry 0 rz 0.01 deg; joints [25.21, -41.968, 95.758, -149.937, 58.288, 164.166]
  MoveL 8917 to (-398.78, -21.15, -9.27) mm, rotated rx 180 ry 0 rz 0.01 deg; joints [24.998, -41.807, 95.454, -150.132, 58.101, 164.21]
  MoveL 8918 to (-397.18, -27.56, -9.51) mm, rotated rx -180 ry 0 rz 0.01 deg; joints [24.813, -41.99, 95.869, -150.412, 58.249, 164.457]
  MoveL 8919 to (-390.67, -28.66, -9.76) mm, rotated rx -180 ry 0 rz 0.01 deg; joints [24.876, -42.283, 96.504, -150.444, 58.564, 164.617]
  MoveL 8920 to (-387.05, -23.13, -10) mm, rotated rx -180 ry 0 rz 0.01 deg; joints [25.114, -42.321, 96.597, -150.194, 58.68, 164.508]
  MoveC 8921 to (-388.69, -19.16, -10) mm, rotated rx -180 ry 0 rz 0.01 deg; joints [25.219, -42.173, 96.281, -150.026, 58.566, 164.348] to (-392.66, -17.52, -10) mm, rotated rx 180 ry 0 rz 0.01 deg; joints [25.211, -41.968, 95.854, -149.966, 58.371, 164.221]
  MoveC 8922 to (-396.62, -19.16, -10) mm, rotated rx 180 ry 0 rz 0.01 deg; joints [25.097, -41.827, 95.564, -150.049, 58.208, 164.203] to (-398.26, -23.13, -10) mm, rotated rx 180 ry 0 rz 0.01 deg; joints [24.942, -41.833, 95.583, -150.227, 58.174, 164.304]
  MoveL 8923 to (-398.26, -23.64, -10) mm, rotated rx 180 ry 0 rz 0.01 deg; joints [24.925, -41.843, 95.604, -150.249, 58.179, 164.321]
  MoveC 8924 to (-397.65, -25.13, -10) mm, rotated rx 180 ry 0 rz 0.01 deg; joints [24.885, -41.899, 95.724, -150.313, 58.222, 164.382] to (-396.15, -25.75, -10) mm, rotated rx 180 ry 0 rz 0.01 deg; joints [24.888, -41.976, 95.885, -150.336, 58.296, 164.429]
  MoveL 8925 to (-394.25, -25.75, -10) mm, rotated rx 180 ry 0 rz 0.01 deg; joints [24.917, -42.059, 96.058, -150.331, 58.382, 164.464]
  MoveC 8926 to (-392.49, -24.65, -10) mm, rotated rx 180 ry 0 rz 0.01 deg; joints [24.98, -42.115, 96.171, -150.277, 58.451, 164.459] to (-392.72, -22.58, -10) mm, rotated rx -180 ry 0 rz 0.01 deg; joints [25.045, -42.064, 96.062, -150.187, 58.419, 164.387]
  MoveL 8927 to (-395.32, -19.32, -10) mm, rotated rx -180 ry 0 rz 0.01 deg; joints [25.112, -41.887, 95.689, -150.052, 58.268, 164.232]
  MoveC 8928 to (-397.16, -18.8, -10) mm, rotated rx 180 ry 0 rz 0.01 deg; joints [25.101, -41.797, 95.5, -150.034, 58.18, 164.181] to (-398.26, -20.35, -10) mm, rotated rx -180 ry 0 rz 0.01 deg; joints [25.033, -41.779, 95.465, -150.105, 58.146, 164.212]
  MoveL 8929 to (-398.26, -23.13, -10) mm, rotated rx 180 ry 0 rz 0.01 deg; joints [24.942, -41.833, 95.583, -150.227, 58.174, 164.304]
  MoveL 8930 to (-398.41, -23.65, -10) mm, rotated rx 180 ry 0 rz 0.01 deg; joints [24.922, -41.837, 95.592, -150.25, 58.172, 164.319]
  MoveL 8931 to (-401.46, -28.61, -10) mm, rotated rx 180 ry 0 rz 0.01 deg; joints [24.713, -41.799, 95.522, -150.476, 58.084, 164.427]
  MoveC 8932 to (-402.31, -29.09, -10) mm, rotated rx 180 ry 0 rz 0.01 deg; joints [24.685, -41.771, 95.465, -150.499, 58.05, 164.427] to (-403.17, -28.62, -10) mm, rotated rx -180 ry 0 rz 0.01 deg; joints [24.688, -41.724, 95.367, -150.48, 58.006, 164.396]
  MoveL 8933 to (-403.27, -28.44, -10) mm, rotated rx 180 ry 0 rz 0.01 deg; joints [24.692, -41.716, 95.35, -150.473, 58, 164.388]
  MoveL 8934 to (-403.58, -27.62, -10) mm, rotated rx 180 ry 0 rz 0.01 deg; joints [24.714, -41.687, 95.287, -150.438, 57.977, 164.355]
  MoveL 8935 to (-403.78, -26.41, -10) mm, rotated rx 180 ry 0 rz 0.01 deg; joints [24.751, -41.655, 95.219, -150.385, 57.956, 164.312]
  MoveL 8936 to (-403.78, 7.61, -10) mm, rotated rx 180 ry 0 rz 0.01 deg; joints [25.855, -40.975, 93.747, -148.889, 57.608, 163.163]
  MoveL 8937 to (-399.89, -2.5, -10) mm, rotated rx 180 ry 0 rz 0.01 deg; joints [25.589, -41.353, 94.549, -149.325, 57.889, 163.583]
  MoveL 8938 to (-399.67, -2.97, -10) mm, rotated rx -180 ry 0 rz 0.01 deg; joints [25.577, -41.372, 94.589, -149.345, 57.904, 163.603]
  MoveL 8939 to (-395.6, -10.08, -10) mm, rotated rx 180 ry 0 rz 0.01 deg; joints [25.409, -41.693, 95.269, -149.648, 58.162, 163.919]
  MoveL 8940 to (-395.3, -10.52, -10) mm, rotated rx -180 ry 0 rz 0.01 deg; joints [25.399, -41.715, 95.314, -149.666, 58.179, 163.939]
  MoveL 8941 to (-387.53, -20.25, -10) mm, rotated rx 180 ry 0 rz 0.01 deg; joints [25.201, -42.245, 96.432, -150.07, 58.63, 164.404]
  MoveL 8942 to (-387.3, -20.5, -10) mm, rotated rx 180 ry 0 rz 0.01 deg; joints [25.197, -42.259, 96.463, -150.08, 58.642, 164.417]
  MoveL 8943 to (-386.61, -21.21, -10) mm, rotated rx 180 ry 0 rz 0.01 deg; joints [25.184, -42.303, 96.556, -150.109, 58.681, 164.453]
  MoveL 8944 to (-386.07, -21.66, -10) mm, rotated rx 180 ry 0 rz 0.01 deg; joints [25.177, -42.335, 96.624, -150.127, 58.71, 164.477]
  MoveL 8945 to (-376.24, -28.22, -10) mm, rotated rx 180 ry 0 rz 0.01 deg; joints [25.113, -42.884, 97.777, -150.379, 59.216, 164.865]
  MoveL 8946 to (-376.07, -28.32, -10) mm, rotated rx 180 ry 0 rz 0.01 deg; joints [25.112, -42.893, 97.796, -150.383, 59.224, 164.871]
  MoveL 8947 to (-374.91, -29.01, -10) mm, rotated rx 180 ry 0 rz 0.01 deg; joints [25.108, -42.956, 97.928, -150.409, 59.283, 164.914]
  MoveL 8948 to (-374.14, -29.34, -10) mm, rotated rx 180 ry 0 rz 0.01 deg; joints [25.109, -42.995, 98.01, -150.42, 59.321, 164.938]
  MoveL 8949 to (-367.51, -31.27, -10) mm, rotated rx 180 ry 0 rz 0.01 deg; joints [25.148, -43.314, 98.677, -150.477, 59.635, 165.114]
  MoveL 8950 to (-398.96, -31.27, -10) mm, rotated rx -180 ry 0 rz 0.01 deg; joints [24.664, -41.96, 95.861, -150.586, 58.224, 164.56]
  MoveL 8951 to (-399.88, -31.14, -10) mm, rotated rx -180 ry 0 rz 0.01 deg; joints [24.654, -41.917, 95.772, -150.583, 58.181, 164.539]
  MoveL 8952 to (-400.74, -30.86, -10) mm, rotated rx 180 ry 0 rz 0.01 deg; joints [24.651, -41.874, 95.682, -150.573, 58.139, 164.514]
  MoveL 8953 to (-401.19, -30.62, -10) mm, rotated rx -180 ry 0 rz 0.01 deg; joints [24.652, -41.85, 95.632, -150.563, 58.117, 164.498]
  MoveL 8954 to (-401.26, -29.55, -10) mm, rotated rx 180 ry 0 rz 0.01 deg; joints [24.686, -41.826, 95.58, -150.517, 58.103, 164.462]
  MoveL 8955 to (-398.55, -27.51, -10) mm, rotated rx 180 ry 0 rz 0.01 deg; joints [24.794, -41.906, 95.742, -150.42, 58.205, 164.444]
  MoveL 8956 to (-393.93, -23.87, -10) mm, rotated rx -180 ry 0 rz 0.01 deg; joints [24.984, -42.037, 96.008, -150.248, 58.378, 164.408]
  MoveL 8957 to (-392.18, -23.28, -10) mm, rotated rx -180 ry 0 rz 0.01 deg; joints [25.03, -42.102, 96.141, -150.216, 58.451, 164.42]
  MoveL 8958 to (-391.93, -22.79, -10) mm, rotated rx 180 ry 0 rz 0.01 deg; joints [25.05, -42.103, 96.143, -150.194, 58.457, 164.408]
  MoveL 8959 to (-397.13, -18.72, -10.24) mm, rotated rx 180 ry 0 rz 0.01 deg; joints [25.104, -41.785, 95.499, -150.033, 58.19, 164.185]
  MoveL 8960 to (-402.94, -21.84, -10.49) mm, rotated rx -180 ry 0 rz 0.01 deg; joints [24.913, -41.579, 95.101, -150.188, 57.967, 164.188]
  MoveL 8961 to (-402.41, -28.42, -10.73) mm, rotated rx -180 ry 0 rz 0.01 deg; joints [24.706, -41.719, 95.426, -150.479, 58.068, 164.422]
  MoveL 8962 to (-396.17, -30.58, -10.98) mm, rotated rx 180 ry 0 rz 0.01 deg; joints [24.73, -42.022, 96.083, -150.561, 58.383, 164.613]
  MoveL 8963 to (-391.69, -25.73, -11.22) mm, rotated rx 180 ry 0 rz 0.01 deg; joints [24.958, -42.112, 96.284, -150.338, 58.546, 164.541]
  MoveL 8964 to (-394.34, -19.68, -11.46) mm, rotated rx -180 ry 0 rz 0.01 deg; joints [25.116, -41.867, 95.789, -150.084, 58.374, 164.3]
  MoveL 8965 to (-400.94, -19.67, -11.71) mm, rotated rx -180 ry 0 rz 0.01 deg; joints [25.015, -41.567, 95.188, -150.105, 58.084, 164.184]
  MoveL 8966 to (-403.59, -25.72, -11.95) mm, rotated rx -180 ry 0 rz 0.01 deg; joints [24.777, -41.556, 95.201, -150.379, 58.034, 164.342]
  MoveL 8967 to (-399.12, -30.57, -12.2) mm, rotated rx -180 ry 0 rz 0.01 deg; joints [24.686, -41.834, 95.811, -150.584, 58.297, 164.59]
  MoveL 8968 to (-392.88, -28.43, -12.44) mm, rotated rx 180 ry 0 rz 0.01 deg; joints [24.851, -42.053, 96.287, -150.476, 58.568, 164.639]
  MoveL 8969 to (-392.34, -21.85, -12.68) mm, rotated rx 180 ry 0 rz 0.01 deg; joints [25.076, -41.938, 96.059, -150.189, 58.535, 164.44]
  MoveL 8970 to (-398.15, -18.72, -12.93) mm, rotated rx -180 ry 0 rz 0.01 deg; joints [25.09, -41.612, 95.398, -150.071, 58.249, 164.236]
  MoveL 8971 to (-403.35, -22.78, -13.17) mm, rotated rx -180 ry 0 rz 0.01 deg; joints [24.878, -41.452, 95.095, -150.266, 58.063, 164.28]
  MoveL 8972 to (-401.72, -29.17, -13.41) mm, rotated rx -180 ry 0 rz 0.01 deg; joints [24.693, -41.636, 95.513, -150.545, 58.212, 164.528]
  MoveL 8973 to (-395.21, -30.25, -13.66) mm, rotated rx -180 ry 0 rz 0.01 deg; joints [24.757, -41.929, 96.149, -150.578, 58.529, 164.688]
  MoveL 8974 to (-391.61, -24.71, -13.9) mm, rotated rx -180 ry 0 rz 0.01 deg; joints [24.994, -41.967, 96.241, -150.328, 58.645, 164.578]
  MoveL 8975 to (-395.24, -19.2, -14.15) mm, rotated rx 180 ry 0 rz 0.01 deg; joints [25.12, -41.69, 95.679, -150.101, 58.433, 164.337]
  MoveL 8976 to (-401.74, -20.3, -14.39) mm, rotated rx -180 ry 0 rz 0.01 deg; joints [24.984, -41.416, 95.134, -150.169, 58.158, 164.26]
  MoveL 8977 to (-403.34, -26.71, -14.63) mm, rotated rx 180 ry 0 rz 0.01 deg; joints [24.75, -41.459, 95.258, -150.457, 58.16, 164.448]
  MoveL 8978 to (-398.12, -30.74, -14.88) mm, rotated rx -180 ry 0 rz 0.01 deg; joints [24.697, -41.753, 95.902, -150.623, 58.45, 164.683]
  MoveL 8979 to (-392.32, -27.57, -15.12) mm, rotated rx -180 ry 0 rz 0.01 deg; joints [24.89, -41.932, 96.293, -150.471, 58.69, 164.69]
  MoveL 8980 to (-392.9, -21, -15.37) mm, rotated rx 180 ry 0 rz 0.01 deg; joints [25.097, -41.769, 95.964, -150.189, 58.606, 164.471]
  MoveL 8981 to (-399.15, -18.89, -15.61) mm, rotated rx -180 ry 0 rz 0.01 deg; joints [25.071, -41.444, 95.306, -150.117, 58.309, 164.292]
  MoveL 8982 to (-403.6, -23.77, -15.85) mm, rotated rx 180 ry 0 rz 0.01 deg; joints [24.844, -41.332, 95.107, -150.345, 58.166, 164.378]
  MoveL 8983 to (-400.91, -29.8, -16.1) mm, rotated rx 180 ry 0 rz 0.01 deg; joints [24.687, -41.554, 95.604, -150.605, 58.36, 164.632]
  MoveL 8984 to (-394.31, -29.76, -16.34) mm, rotated rx -180 ry 0 rz 0.01 deg; joints [24.788, -41.829, 96.201, -150.588, 58.67, 164.757]
  MoveL 8985 to (-391.7, -23.69, -16.59) mm, rotated rx 180 ry 0 rz 0.01 deg; joints [25.028, -41.814, 96.182, -150.318, 58.736, 164.612]
  MoveL 8986 to (-396.2, -18.87, -16.83) mm, rotated rx 180 ry 0 rz 0.01 deg; joints [25.117, -41.513, 95.569, -150.124, 58.491, 164.378]
  MoveL 8987 to (-402.43, -21.06, -17.07) mm, rotated rx 180 ry 0 rz 0.01 deg; joints [24.951, -41.273, 95.095, -150.239, 58.239, 164.341]
  MoveL 8988 to (-402.93, -27.64, -17.32) mm, rotated rx -180 ry 0 rz 0.01 deg; joints [24.728, -41.367, 95.326, -150.532, 58.294, 164.555]
  MoveL 8989 to (-397.09, -30.73, -17.56) mm, rotated rx 180 ry 0 rz 0.01 deg; joints [24.715, -41.668, 95.986, -150.655, 58.601, 164.769]
  MoveL 8990 to (-391.92, -26.64, -17.8) mm, rotated rx 180 ry 0 rz 0.01 deg; joints [24.928, -41.802, 96.282, -150.463, 58.804, 164.735]
  MoveL 8991 to (-393.6, -20.25, -18.05) mm, rotated rx -180 ry 0 rz 0.01 deg; joints [25.113, -41.595, 95.86, -150.193, 58.671, 164.502]
  MoveL 8992 to (-400.12, -19.23, -18.29) mm, rotated rx -180 ry 0 rz 0.01 deg; joints [25.046, -41.28, 95.224, -150.169, 58.373, 164.354]
  MoveL 8993 to (-403.67, -24.79, -18.54) mm, rotated rx -180 ry 0 rz 0.01 deg; joints [24.811, -41.22, 95.134, -150.424, 58.277, 164.478]
  MoveL 8994 to (-400.01, -30.28, -18.78) mm, rotated rx 180 ry 0 rz 0.01 deg; joints [24.686, -41.474, 95.698, -150.658, 58.512, 164.732]
  MoveL 8995 to (-393.51, -29.12, -19.02) mm, rotated rx 180 ry 0 rz 0.01 deg; joints [24.823, -41.722, 96.238, -150.592, 58.805, 164.819]
  MoveL 8996 to (-391.96, -22.71, -19.27) mm, rotated rx -180 ry 0 rz 0.01 deg; joints [25.058, -41.654, 96.108, -150.31, 58.819, 164.644]
  MoveL 8997 to (-397.21, -18.71, -19.51) mm, rotated rx 180 ry 0 rz 0.01 deg; joints [25.109, -41.338, 95.462, -150.154, 58.547, 164.423]
  MoveL 8998 to (-402.98, -21.92, -19.76) mm, rotated rx -180 ry 0 rz 0.01 deg; joints [24.916, -41.137, 95.072, -150.313, 58.327, 164.427]
  MoveL 8999 to (-402.36, -28.49, -20) mm, rotated rx -180 ry 0 rz 0.01 deg; joints [24.71, -41.279, 95.405, -150.602, 58.433, 164.661]
  MoveC 9000 to (-398.6, -30.56, -20) mm, rotated rx -180 ry 0 rz 0.01 deg; joints [24.699, -41.482, 95.833, -150.682, 58.627, 164.798] to (-394.48, -29.38, -20) mm, rotated rx -180 ry 0 rz 0.01 deg; joints [24.801, -41.638, 96.158, -150.618, 58.802, 164.834]
  MoveC 9001 to (-392.4, -25.62, -20) mm, rotated rx 180 ry 0 rz 0.01 deg; joints [24.956, -41.656, 96.188, -150.448, 58.857, 164.749] to (-393.59, -21.5, -20) mm, rotated rx -180 ry 0 rz 0.01 deg; joints [25.073, -41.525, 95.907, -150.272, 58.76, 164.593]
  MoveL 9002 to (-395.33, -19.32, -20) mm, rotated rx -180 ry 0 rz 0.01 deg; joints [25.118, -41.408, 95.658, -150.182, 58.659, 164.49]
  MoveC 9003 to (-397.16, -18.8, -20) mm, rotated rx -180 ry 0 rz 0.01 deg; joints [25.107, -41.318, 95.468, -150.164, 58.569, 164.439] to (-398.27, -20.35, -20) mm, rotated rx -180 ry 0 rz 0.01 deg; joints [25.039, -41.3, 95.434, -150.235, 58.535, 164.47]
  MoveL 9004 to (-398.27, -23.64, -20) mm, rotated rx -180 ry 0 rz 0.01 deg; joints [24.931, -41.364, 95.573, -150.379, 58.57, 164.578]
  MoveC 9005 to (-397.65, -25.14, -20) mm, rotated rx -180 ry 0 rz 0.01 deg; joints [24.892, -41.42, 95.693, -150.442, 58.614, 164.638] to (-396.15, -25.76, -20) mm, rotated rx -180 ry 0 rz 0.01 deg; joints [24.894, -41.496, 95.854, -150.465, 58.688, 164.686]
  MoveL 9006 to (-394.26, -25.76, -20) mm, rotated rx -180 ry 0 rz 0.01 deg; joints [24.923, -41.578, 96.026, -150.46, 58.775, 164.72]
  MoveC 9007 to (-392.5, -24.65, -20) mm, rotated rx -180 ry 0 rz 0.01 deg; joints [24.986, -41.633, 96.139, -150.406, 58.843, 164.716] to (-392.73, -22.58, -20) mm, rotated rx 180 ry 0 rz 0.01 deg; joints [25.051, -41.583, 96.031, -150.316, 58.811, 164.644]
  MoveL 9008 to (-393.59, -21.5, -20) mm, rotated rx -180 ry 0 rz 0.01 deg; joints [25.073, -41.525, 95.907, -150.272, 58.76, 164.593]
  MoveC 9009 to (-394.36, -21.12, -20) mm, rotated rx -180 ry 0 rz 0.01 deg; joints [25.074, -41.485, 95.821, -150.258, 58.721, 164.567] to (-395.14, -21.48, -20) mm, rotated rx 180 ry 0 rz 0.01 deg; joints [25.05, -41.458, 95.766, -150.276, 58.69, 164.564]
  MoveL 9010 to (-401.47, -29.1, -20) mm, rotated rx 180 ry 0 rz 0.01 deg; joints [24.704, -41.329, 95.511, -150.626, 58.48, 164.698]
  MoveL 9011 to (-401.19, -30.62, -20) mm, rotated rx 180 ry 0 rz 0.01 deg; joints [24.658, -41.371, 95.6, -150.692, 58.509, 164.752]
  MoveL 9012 to (-400.74, -30.86, -20) mm, rotated rx 180 ry 0 rz 0.01 deg; joints [24.657, -41.395, 95.651, -150.701, 58.532, 164.768]
  MoveL 9013 to (-399.88, -31.14, -20) mm, rotated rx -180 ry 0 rz 0.01 deg; joints [24.661, -41.437, 95.741, -150.711, 58.574, 164.793]
  MoveL 9014 to (-398.96, -31.27, -20) mm, rotated rx 180 ry 0 rz 0.01 deg; joints [24.67, -41.48, 95.83, -150.714, 58.617, 164.814]
  MoveL 9015 to (-367.62, -31.27, -20) mm, rotated rx 180 ry 0 rz 0.01 deg; joints [25.153, -42.819, 98.636, -150.602, 60.032, 165.37]
  MoveL 9016 to (-373.86, -29.45, -20) mm, rotated rx -180 ry 0 rz 0.01 deg; joints [25.116, -42.521, 98.009, -150.549, 59.734, 165.204]
  MoveL 9017 to (-374.35, -29.26, -20) mm, rotated rx -180 ry 0 rz 0.01 deg; joints [25.114, -42.497, 97.957, -150.543, 59.71, 165.189]
  MoveL 9018 to (-375.36, -28.78, -20) mm, rotated rx 180 ry 0 rz 0.01 deg; joints [25.114, -42.445, 97.848, -150.526, 59.66, 165.156]
  MoveL 9019 to (-375.81, -28.53, -20) mm, rotated rx 180 ry 0 rz 0.01 deg; joints [25.116, -42.422, 97.798, -150.517, 59.637, 165.14]
  MoveL 9020 to (-386.07, -21.65, -20) mm, rotated rx -180 ry 0 rz 0.01 deg; joints [25.184, -41.852, 96.592, -150.255, 59.103, 164.735]
  MoveL 9021 to (-386.58, -21.23, -20) mm, rotated rx -180 ry 0 rz 0.01 deg; joints [25.19, -41.822, 96.528, -150.238, 59.075, 164.712]
  MoveL 9022 to (-387.29, -20.52, -20) mm, rotated rx 180 ry 0 rz 0.01 deg; joints [25.202, -41.778, 96.434, -150.21, 59.036, 164.676]
  MoveL 9023 to (-387.54, -20.24, -20) mm, rotated rx 180 ry 0 rz 0.01 deg; joints [25.207, -41.762, 96.4, -150.198, 59.022, 164.663]
  MoveL 9024 to (-395.31, -10.51, -20) mm, rotated rx 180 ry 0 rz 0.01 deg; joints [25.406, -41.237, 95.283, -149.797, 58.567, 164.2]
  MoveL 9025 to (-395.6, -10.08, -20) mm, rotated rx 180 ry 0 rz 0.01 deg; joints [25.415, -41.215, 95.238, -149.779, 58.549, 164.18]
  MoveL 9026 to (-399.67, -2.97, -20) mm, rotated rx 180 ry 0 rz 0.01 deg; joints [25.583, -40.897, 94.558, -149.479, 58.288, 163.866]
  MoveL 9027 to (-399.88, -2.51, -20) mm, rotated rx -180 ry 0 rz 0.01 deg; joints [25.595, -40.878, 94.519, -149.46, 58.273, 163.846]
  MoveL 9028 to (-403.78, 7.53, -20) mm, rotated rx 180 ry 0 rz 0.01 deg; joints [25.858, -40.504, 93.72, -149.029, 57.988, 163.431]
  MoveL 9029 to (-403.78, -26.41, -20) mm, rotated rx 180 ry 0 rz 0.01 deg; joints [24.757, -41.177, 95.188, -150.515, 58.346, 164.567]
  MoveL 9030 to (-403.58, -27.62, -20) mm, rotated rx 180 ry 0 rz 0.01 deg; joints [24.72, -41.209, 95.256, -150.567, 58.368, 164.61]
  MoveL 9031 to (-403.27, -28.44, -20) mm, rotated rx -180 ry 0 rz 0.01 deg; joints [24.698, -41.238, 95.319, -150.602, 58.391, 164.643]
  Set speed (500.0 mm/s)
  MoveL 9032 to (-403.27, -28.44, 11) mm, rotated rx 180 ry 0 rz 0.01 deg; joints [24.679, -42.707, 95.389, -150.188, 57.168, 163.838]
  Set speed (500.0 mm/s)
  MoveL 9033 to (-399.07, -22.37, 11) mm, rotated rx -180 ry 0 rz 0.01 deg; joints [24.941, -42.775, 95.516, -149.91, 57.299, 163.709]
  Set speed (100.0 mm/s)
  MoveL 9034 to (-399.07, -22.37, -8.23) mm, rotated rx -180 ry 0 rz 0.01 deg; joints [24.953, -41.867, 95.482, -150.172, 58.06, 164.218]
  MoveL 9035 to (-399.09, -22.53, -8.85) mm, rotated rx -180 ry 0 rz 0.01 deg; joints [24.948, -41.84, 95.486, -150.188, 58.085, 164.239]
  MoveL 9036 to (-399.12, -22.98, -9.32) mm, rotated rx -180 ry 0 rz 0.01 deg; joints [24.933, -41.825, 95.501, -150.213, 58.107, 164.266]
  MoveL 9037 to (-399.11, -23.59, -9.5) mm, rotated rx 180 ry 0 rz 0.01 deg; joints [24.913, -41.829, 95.527, -150.243, 58.121, 164.291]
  MoveL 9038 to (-395.08, -28.83, -9.74) mm, rotated rx -180 ry 0 rz 0.01 deg; joints [24.803, -42.095, 96.112, -150.465, 58.366, 164.543]
  MoveL 9039 to (-388.67, -27.24, -9.99) mm, rotated rx 180 ry 0 rz 0.01 deg; joints [24.953, -42.331, 96.624, -150.379, 58.649, 164.613]
  MoveL 9040 to (-387.56, -20.73, -10.23) mm, rotated rx 180 ry 0 rz 0.01 deg; joints [25.185, -42.242, 96.45, -150.094, 58.642, 164.426]
  MoveL 9041 to (-393.08, -17.1, -10.48) mm, rotated rx -180 ry 0 rz 0.01 deg; joints [25.219, -41.919, 95.797, -149.955, 58.366, 164.212]
  MoveL 9042 to (-398.61, -20.71, -10.72) mm, rotated rx 180 ry 0 rz 0.01 deg; joints [25.016, -41.736, 95.447, -150.131, 58.162, 164.236]
  MoveL 9043 to (-397.53, -27.22, -10.96) mm, rotated rx 180 ry 0 rz 0.01 deg; joints [24.819, -41.898, 95.819, -150.417, 58.287, 164.477]
  MoveL 9044 to (-391.13, -28.84, -11.21) mm, rotated rx -180 ry 0 rz 0.01 deg; joints [24.864, -42.197, 96.466, -150.473, 58.602, 164.652]
  MoveL 9045 to (-387.08, -23.62, -11.45) mm, rotated rx 180 ry 0 rz 0.01 deg; joints [25.098, -42.26, 96.611, -150.235, 58.742, 164.561]
  MoveL 9046 to (-390.23, -17.82, -11.7) mm, rotated rx -180 ry 0 rz 0.01 deg; joints [25.24, -41.998, 96.081, -149.994, 58.55, 164.32]
  MoveL 9047 to (-396.81, -18.39, -11.94) mm, rotated rx 180 ry 0 rz 0.01 deg; joints [25.12, -41.711, 95.509, -150.041, 58.267, 164.224]
  MoveL 9048 to (-398.93, -24.65, -12.18) mm, rotated rx 180 ry 0 rz 0.01 deg; joints [24.883, -41.729, 95.58, -150.324, 58.245, 164.398]
  MoveL 9049 to (-394.05, -29.09, -12.43) mm, rotated rx -180 ry 0 rz 0.01 deg; joints [24.812, -42.016, 96.209, -150.508, 58.521, 164.64]
  MoveL 9050 to (-388.02, -26.4, -12.67) mm, rotated rx 180 ry 0 rz 0.01 deg; joints [24.993, -42.214, 96.64, -150.375, 58.776, 164.666]
  MoveL 9051 to (-388.07, -19.8, -12.92) mm, rotated rx 180 ry 0 rz 0.01 deg; joints [25.21, -42.072, 96.356, -150.09, 58.715, 164.456]
  MoveL 9052 to (-394.14, -17.2, -13.16) mm, rotated rx 180 ry 0 rz 0.01 deg; joints [25.201, -41.746, 95.697, -149.997, 58.424, 164.265]
  MoveL 9053 to (-398.95, -21.72, -13.4) mm, rotated rx -180 ry 0 rz 0.01 deg; joints [24.98, -41.613, 95.451, -150.211, 58.261, 164.333]
  MoveL 9054 to (-396.74, -27.94, -13.65) mm, rotated rx 180 ry 0 rz 0.01 deg; joints [24.809, -41.818, 95.913, -150.481, 58.435, 164.584]
  MoveL 9055 to (-390.15, -28.41, -13.89) mm, rotated rx 180 ry 0 rz 0.01 deg; joints [24.895, -42.101, 96.528, -150.485, 58.748, 164.725]
  MoveL 9056 to (-387.09, -22.56, -14.14) mm, rotated rx 180 ry 0 rz 0.01 deg; joints [25.135, -42.109, 96.558, -150.223, 58.836, 164.596]
  MoveL 9057 to (-391.21, -17.4, -14.38) mm, rotated rx 180 ry 0 rz 0.01 deg; joints [25.24, -41.819, 95.967, -150.014, 58.606, 164.358]
